(* Logix 5000 project; controller reports 1756-L63 rev 20.11; software revision 20.04; part 30 of 52 *)

        [2217].log_data[18].valid := 1, [2217].log_data[19].valid := 1, [2217].time.Year := 2023, [2217].time.Month := 1, [2217].time.Day := 17, [2217].time.Hour := 9, [2217].time.Minute := 9, [2217].time.Second := 59, [2218].log_data[0].min := 1.0, [2218].log_data[0].max := 1.0, [2218].log_data[0].total := 300.0, [2218].log_data[0].time := 300.0, [2218].log_data[0].minminute := 10, [2218].log_data[0].maxminute := 10, [2218].log_data[0].valid := 1, [2218].log_data[1].valid := 1, [2218].log_data[2].valid := 1, [2218].log_data[3].valid := 1, [2218].log_data[4].valid := 1, [2218].log_data[5].valid := 1, [2218].log_data[6].valid := 1, [2218].log_data[7].valid := 1, [2218].log_data[8].valid := 1, [2218].log_data[9].valid := 1, [2218].log_data[10].valid := 1, [2218].log_data[11].valid := 1, [2218].log_data[12].valid := 1, [2218].log_data[13].valid := 1, [2218].log_data[14].valid := 1, [2218].log_data[15].valid := 1, [2218].log_data[16].valid := 1, [2218].log_data[17].valid := 1, [2218].log_data[18].valid := 1, [2218].log_data[19].valid := 1, [2218].time.Year := 2023, [2218].time.Month := 1, [2218].time.Day := 17, [2218].time.Hour := 9, [2218].time.Minute := 14, [2218].time.Second := 59, [2219].log_data[0].min := 1.0, [2219].log_data[0].max := 1.0, [2219].log_data[0].total := 300.0, [2219].log_data[0].time := 300.0, [2219].log_data[0].minminute := 15, [2219].log_data[0].maxminute := 15, [2219].log_data[0].valid := 1, [2219].log_data[1].valid := 1, [2219].log_data[2].valid := 1, [2219].log_data[3].valid := 1, [2219].log_data[4].valid := 1, [2219].log_data[5].valid := 1, [2219].log_data[6].valid := 1, [2219].log_data[7].valid := 1, [2219].log_data[8].valid := 1, [2219].log_data[9].valid := 1, [2219].log_data[10].valid := 1, [2219].log_data[11].valid := 1, [2219].log_data[12].valid := 1, [2219].log_data[13].valid := 1,
        [2219].log_data[14].valid := 1, [2219].log_data[15].valid := 1, [2219].log_data[16].valid := 1, [2219].log_data[17].valid := 1, [2219].log_data[18].valid := 1, [2219].log_data[19].valid := 1, [2219].time.Year := 2023, [2219].time.Month := 1, [2219].time.Day := 17, [2219].time.Hour := 9, [2219].time.Minute := 19, [2219].time.Second := 59, [2220].log_data[0].min := 1.0, [2220].log_data[0].max := 1.0, [2220].log_data[0].total := 300.0, [2220].log_data[0].time := 300.0, [2220].log_data[0].minminute := 20, [2220].log_data[0].maxminute := 20, [2220].log_data[0].valid := 1, [2220].log_data[1].valid := 1, [2220].log_data[2].valid := 1, [2220].log_data[3].valid := 1, [2220].log_data[4].valid := 1, [2220].log_data[5].valid := 1, [2220].log_data[6].valid := 1, [2220].log_data[7].valid := 1, [2220].log_data[8].valid := 1, [2220].log_data[9].valid := 1, [2220].log_data[10].valid := 1, [2220].log_data[11].valid := 1, [2220].log_data[12].valid := 1, [2220].log_data[13].valid := 1, [2220].log_data[14].valid := 1, [2220].log_data[15].valid := 1, [2220].log_data[16].valid := 1, [2220].log_data[17].valid := 1, [2220].log_data[18].valid := 1, [2220].log_data[19].valid := 1, [2220].time.Year := 2023, [2220].time.Month := 1, [2220].time.Day := 17, [2220].time.Hour := 9, [2220].time.Minute := 24, [2220].time.Second := 59, [2221].log_data[0].min := 1.0, [2221].log_data[0].max := 1.0, [2221].log_data[0].total := 300.0, [2221].log_data[0].time := 300.0, [2221].log_data[0].minminute := 25, [2221].log_data[0].maxminute := 25, [2221].log_data[0].valid := 1, [2221].log_data[1].valid := 1, [2221].log_data[2].valid := 1, [2221].log_data[3].valid := 1, [2221].log_data[4].valid := 1, [2221].log_data[5].valid := 1, [2221].log_data[6].valid := 1, [2221].log_data[7].valid := 1, [2221].log_data[8].valid := 1, [2221].log_data[9].valid := 1,
        [2221].log_data[10].valid := 1, [2221].log_data[11].valid := 1, [2221].log_data[12].valid := 1, [2221].log_data[13].valid := 1, [2221].log_data[14].valid := 1, [2221].log_data[15].valid := 1, [2221].log_data[16].valid := 1, [2221].log_data[17].valid := 1, [2221].log_data[18].valid := 1, [2221].log_data[19].valid := 1, [2221].time.Year := 2023, [2221].time.Month := 1, [2221].time.Day := 17, [2221].time.Hour := 9, [2221].time.Minute := 29, [2221].time.Second := 59, [2222].log_data[0].min := 1.0, [2222].log_data[0].max := 1.0, [2222].log_data[0].total := 300.0, [2222].log_data[0].time := 300.0, [2222].log_data[0].minminute := 30, [2222].log_data[0].maxminute := 30, [2222].log_data[0].valid := 1, [2222].log_data[1].valid := 1, [2222].log_data[2].valid := 1, [2222].log_data[3].valid := 1, [2222].log_data[4].valid := 1, [2222].log_data[5].valid := 1, [2222].log_data[6].valid := 1, [2222].log_data[7].valid := 1, [2222].log_data[8].valid := 1, [2222].log_data[9].valid := 1, [2222].log_data[10].valid := 1, [2222].log_data[11].valid := 1, [2222].log_data[12].valid := 1, [2222].log_data[13].valid := 1, [2222].log_data[14].valid := 1, [2222].log_data[15].valid := 1, [2222].log_data[16].valid := 1, [2222].log_data[17].valid := 1, [2222].log_data[18].valid := 1, [2222].log_data[19].valid := 1, [2222].time.Year := 2023, [2222].time.Month := 1, [2222].time.Day := 17, [2222].time.Hour := 9, [2222].time.Minute := 34, [2222].time.Second := 59, [2223].log_data[0].min := 1.0, [2223].log_data[0].max := 1.0, [2223].log_data[0].total := 300.0, [2223].log_data[0].time := 300.0, [2223].log_data[0].minminute := 35, [2223].log_data[0].maxminute := 35, [2223].log_data[0].valid := 1, [2223].log_data[1].valid := 1, [2223].log_data[2].valid := 1, [2223].log_data[3].valid := 1, [2223].log_data[4].valid := 1, [2223].log_data[5].valid := 1,
        [2223].log_data[6].valid := 1, [2223].log_data[7].valid := 1, [2223].log_data[8].valid := 1, [2223].log_data[9].valid := 1, [2223].log_data[10].valid := 1, [2223].log_data[11].valid := 1, [2223].log_data[12].valid := 1, [2223].log_data[13].valid := 1, [2223].log_data[14].valid := 1, [2223].log_data[15].valid := 1, [2223].log_data[16].valid := 1, [2223].log_data[17].valid := 1, [2223].log_data[18].valid := 1, [2223].log_data[19].valid := 1, [2223].time.Year := 2023, [2223].time.Month := 1, [2223].time.Day := 17, [2223].time.Hour := 9, [2223].time.Minute := 39, [2223].time.Second := 59, [2224].log_data[0].min := 1.0, [2224].log_data[0].max := 1.0, [2224].log_data[0].total := 300.0, [2224].log_data[0].time := 300.0, [2224].log_data[0].minminute := 40, [2224].log_data[0].maxminute := 40, [2224].log_data[0].valid := 1, [2224].log_data[1].valid := 1, [2224].log_data[2].valid := 1, [2224].log_data[3].valid := 1, [2224].log_data[4].valid := 1, [2224].log_data[5].valid := 1, [2224].log_data[6].valid := 1, [2224].log_data[7].valid := 1, [2224].log_data[8].valid := 1, [2224].log_data[9].valid := 1, [2224].log_data[10].valid := 1, [2224].log_data[11].valid := 1, [2224].log_data[12].valid := 1, [2224].log_data[13].valid := 1, [2224].log_data[14].valid := 1, [2224].log_data[15].valid := 1, [2224].log_data[16].valid := 1, [2224].log_data[17].valid := 1, [2224].log_data[18].valid := 1, [2224].log_data[19].valid := 1, [2224].time.Year := 2023, [2224].time.Month := 1, [2224].time.Day := 17, [2224].time.Hour := 9, [2224].time.Minute := 44, [2224].time.Second := 59, [2225].log_data[0].min := 1.0, [2225].log_data[0].max := 1.0, [2225].log_data[0].total := 300.0, [2225].log_data[0].time := 300.0, [2225].log_data[0].minminute := 45, [2225].log_data[0].maxminute := 45, [2225].log_data[0].valid := 1, [2225].log_data[1].valid := 1,
        [2225].log_data[2].valid := 1, [2225].log_data[3].valid := 1, [2225].log_data[4].valid := 1, [2225].log_data[5].valid := 1, [2225].log_data[6].valid := 1, [2225].log_data[7].valid := 1, [2225].log_data[8].valid := 1, [2225].log_data[9].valid := 1, [2225].log_data[10].valid := 1, [2225].log_data[11].valid := 1, [2225].log_data[12].valid := 1, [2225].log_data[13].valid := 1, [2225].log_data[14].valid := 1, [2225].log_data[15].valid := 1, [2225].log_data[16].valid := 1, [2225].log_data[17].valid := 1, [2225].log_data[18].valid := 1, [2225].log_data[19].valid := 1, [2225].time.Year := 2023, [2225].time.Month := 1, [2225].time.Day := 17, [2225].time.Hour := 9, [2225].time.Minute := 49, [2225].time.Second := 59, [2226].log_data[0].min := 1.0, [2226].log_data[0].max := 1.0, [2226].log_data[0].total := 300.0, [2226].log_data[0].time := 300.0, [2226].log_data[0].minminute := 50, [2226].log_data[0].maxminute := 50, [2226].log_data[0].valid := 1, [2226].log_data[1].valid := 1, [2226].log_data[2].valid := 1, [2226].log_data[3].valid := 1, [2226].log_data[4].valid := 1, [2226].log_data[5].valid := 1, [2226].log_data[6].valid := 1, [2226].log_data[7].valid := 1, [2226].log_data[8].valid := 1, [2226].log_data[9].valid := 1, [2226].log_data[10].valid := 1, [2226].log_data[11].valid := 1, [2226].log_data[12].valid := 1, [2226].log_data[13].valid := 1, [2226].log_data[14].valid := 1, [2226].log_data[15].valid := 1, [2226].log_data[16].valid := 1, [2226].log_data[17].valid := 1, [2226].log_data[18].valid := 1, [2226].log_data[19].valid := 1, [2226].time.Year := 2023, [2226].time.Month := 1, [2226].time.Day := 17, [2226].time.Hour := 9, [2226].time.Minute := 54, [2226].time.Second := 59, [2227].log_data[0].min := 1.0, [2227].log_data[0].max := 1.0, [2227].log_data[0].total := 300.0, [2227].log_data[0].time := 300.0,
        [2227].log_data[0].minminute := 55, [2227].log_data[0].maxminute := 55, [2227].log_data[0].valid := 1, [2227].log_data[1].valid := 1, [2227].log_data[2].valid := 1, [2227].log_data[3].valid := 1, [2227].log_data[4].valid := 1, [2227].log_data[5].valid := 1, [2227].log_data[6].valid := 1, [2227].log_data[7].valid := 1, [2227].log_data[8].valid := 1, [2227].log_data[9].valid := 1, [2227].log_data[10].valid := 1, [2227].log_data[11].valid := 1, [2227].log_data[12].valid := 1, [2227].log_data[13].valid := 1, [2227].log_data[14].valid := 1, [2227].log_data[15].valid := 1, [2227].log_data[16].valid := 1, [2227].log_data[17].valid := 1, [2227].log_data[18].valid := 1, [2227].log_data[19].valid := 1, [2227].time.Year := 2023, [2227].time.Month := 1, [2227].time.Day := 17, [2227].time.Hour := 9, [2227].time.Minute := 59, [2227].time.Second := 59, [2228].log_data[0].min := 1.0, [2228].log_data[0].max := 1.0, [2228].log_data[0].total := 300.0, [2228].log_data[0].time := 300.0, [2228].log_data[0].valid := 1, [2228].log_data[1].valid := 1, [2228].log_data[2].valid := 1, [2228].log_data[3].valid := 1, [2228].log_data[4].valid := 1, [2228].log_data[5].valid := 1, [2228].log_data[6].valid := 1, [2228].log_data[7].valid := 1, [2228].log_data[8].valid := 1, [2228].log_data[9].valid := 1, [2228].log_data[10].valid := 1, [2228].log_data[11].valid := 1, [2228].log_data[12].valid := 1, [2228].log_data[13].valid := 1, [2228].log_data[14].valid := 1, [2228].log_data[15].valid := 1, [2228].log_data[16].valid := 1, [2228].log_data[17].valid := 1, [2228].log_data[18].valid := 1, [2228].log_data[19].valid := 1, [2228].time.Year := 2023, [2228].time.Month := 1, [2228].time.Day := 17, [2228].time.Hour := 10, [2228].time.Minute := 4, [2228].time.Second := 59, [2229].log_data[0].min := 1.0, [2229].log_data[0].max := 1.0,
        [2229].log_data[0].total := 300.0, [2229].log_data[0].time := 300.0, [2229].log_data[0].minminute := 5, [2229].log_data[0].maxminute := 5, [2229].log_data[0].valid := 1, [2229].log_data[1].valid := 1, [2229].log_data[2].valid := 1, [2229].log_data[3].valid := 1, [2229].log_data[4].valid := 1, [2229].log_data[5].valid := 1, [2229].log_data[6].valid := 1, [2229].log_data[7].valid := 1, [2229].log_data[8].valid := 1, [2229].log_data[9].valid := 1, [2229].log_data[10].valid := 1, [2229].log_data[11].valid := 1, [2229].log_data[12].valid := 1, [2229].log_data[13].valid := 1, [2229].log_data[14].valid := 1, [2229].log_data[15].valid := 1, [2229].log_data[16].valid := 1, [2229].log_data[17].valid := 1, [2229].log_data[18].valid := 1, [2229].log_data[19].valid := 1, [2229].time.Year := 2023, [2229].time.Month := 1, [2229].time.Day := 17, [2229].time.Hour := 10, [2229].time.Minute := 9, [2229].time.Second := 59, [2230].log_data[0].min := 1.0, [2230].log_data[0].max := 1.0, [2230].log_data[0].total := 300.0, [2230].log_data[0].time := 300.0, [2230].log_data[0].minminute := 10, [2230].log_data[0].maxminute := 10, [2230].log_data[0].valid := 1, [2230].log_data[1].valid := 1, [2230].log_data[2].valid := 1, [2230].log_data[3].valid := 1, [2230].log_data[4].valid := 1, [2230].log_data[5].valid := 1, [2230].log_data[6].valid := 1, [2230].log_data[7].valid := 1, [2230].log_data[8].valid := 1, [2230].log_data[9].valid := 1, [2230].log_data[10].valid := 1, [2230].log_data[11].valid := 1, [2230].log_data[12].valid := 1, [2230].log_data[13].valid := 1, [2230].log_data[14].valid := 1, [2230].log_data[15].valid := 1, [2230].log_data[16].valid := 1, [2230].log_data[17].valid := 1, [2230].log_data[18].valid := 1, [2230].log_data[19].valid := 1, [2230].time.Year := 2023, [2230].time.Month := 1, [2230].time.Day := 17, [2230].time.Hour := 10,
        [2230].time.Minute := 14, [2230].time.Second := 59, [2231].log_data[0].min := 1.0, [2231].log_data[0].max := 1.0, [2231].log_data[0].total := 300.0, [2231].log_data[0].time := 300.0, [2231].log_data[0].minminute := 15, [2231].log_data[0].maxminute := 15, [2231].log_data[0].valid := 1, [2231].log_data[1].valid := 1, [2231].log_data[2].valid := 1, [2231].log_data[3].valid := 1, [2231].log_data[4].valid := 1, [2231].log_data[5].valid := 1, [2231].log_data[6].valid := 1, [2231].log_data[7].valid := 1, [2231].log_data[8].valid := 1, [2231].log_data[9].valid := 1, [2231].log_data[10].valid := 1, [2231].log_data[11].valid := 1, [2231].log_data[12].valid := 1, [2231].log_data[13].valid := 1, [2231].log_data[14].valid := 1, [2231].log_data[15].valid := 1, [2231].log_data[16].valid := 1, [2231].log_data[17].valid := 1, [2231].log_data[18].valid := 1, [2231].log_data[19].valid := 1, [2231].time.Year := 2023, [2231].time.Month := 1, [2231].time.Day := 17, [2231].time.Hour := 10, [2231].time.Minute := 19, [2231].time.Second := 59, [2232].log_data[0].min := 1.0, [2232].log_data[0].max := 1.0, [2232].log_data[0].total := 300.0, [2232].log_data[0].time := 300.0, [2232].log_data[0].minminute := 20, [2232].log_data[0].maxminute := 20, [2232].log_data[0].valid := 1, [2232].log_data[1].valid := 1, [2232].log_data[2].valid := 1, [2232].log_data[3].valid := 1, [2232].log_data[4].valid := 1, [2232].log_data[5].valid := 1, [2232].log_data[6].valid := 1, [2232].log_data[7].valid := 1, [2232].log_data[8].valid := 1, [2232].log_data[9].valid := 1, [2232].log_data[10].valid := 1, [2232].log_data[11].valid := 1, [2232].log_data[12].valid := 1, [2232].log_data[13].valid := 1, [2232].log_data[14].valid := 1, [2232].log_data[15].valid := 1, [2232].log_data[16].valid := 1, [2232].log_data[17].valid := 1, [2232].log_data[18].valid := 1, [2232].log_data[19].valid := 1,
        [2232].time.Year := 2023, [2232].time.Month := 1, [2232].time.Day := 17, [2232].time.Hour := 10, [2232].time.Minute := 24, [2232].time.Second := 59, [2233].log_data[0].min := 1.0, [2233].log_data[0].max := 1.0, [2233].log_data[0].total := 300.0, [2233].log_data[0].time := 300.0, [2233].log_data[0].minminute := 25, [2233].log_data[0].maxminute := 25, [2233].log_data[0].valid := 1, [2233].log_data[1].valid := 1, [2233].log_data[2].valid := 1, [2233].log_data[3].valid := 1, [2233].log_data[4].valid := 1, [2233].log_data[5].valid := 1, [2233].log_data[6].valid := 1, [2233].log_data[7].valid := 1, [2233].log_data[8].valid := 1, [2233].log_data[9].valid := 1, [2233].log_data[10].valid := 1, [2233].log_data[11].valid := 1, [2233].log_data[12].valid := 1, [2233].log_data[13].valid := 1, [2233].log_data[14].valid := 1, [2233].log_data[15].valid := 1, [2233].log_data[16].valid := 1, [2233].log_data[17].valid := 1, [2233].log_data[18].valid := 1, [2233].log_data[19].valid := 1, [2233].time.Year := 2023, [2233].time.Month := 1, [2233].time.Day := 17, [2233].time.Hour := 10, [2233].time.Minute := 29, [2233].time.Second := 59, [2234].log_data[0].min := 1.0, [2234].log_data[0].max := 1.0, [2234].log_data[0].total := 300.0, [2234].log_data[0].time := 300.0, [2234].log_data[0].minminute := 30, [2234].log_data[0].maxminute := 30, [2234].log_data[0].valid := 1, [2234].log_data[1].valid := 1, [2234].log_data[2].valid := 1, [2234].log_data[3].valid := 1, [2234].log_data[4].valid := 1, [2234].log_data[5].valid := 1, [2234].log_data[6].valid := 1, [2234].log_data[7].valid := 1, [2234].log_data[8].valid := 1, [2234].log_data[9].valid := 1, [2234].log_data[10].valid := 1, [2234].log_data[11].valid := 1, [2234].log_data[12].valid := 1, [2234].log_data[13].valid := 1, [2234].log_data[14].valid := 1, [2234].log_data[15].valid := 1,
        [2234].log_data[16].valid := 1, [2234].log_data[17].valid := 1, [2234].log_data[18].valid := 1, [2234].log_data[19].valid := 1, [2234].time.Year := 2023, [2234].time.Month := 1, [2234].time.Day := 17, [2234].time.Hour := 10, [2234].time.Minute := 34, [2234].time.Second := 59, [2235].log_data[0].min := 1.0, [2235].log_data[0].max := 1.0, [2235].log_data[0].total := 300.0, [2235].log_data[0].time := 300.0, [2235].log_data[0].minminute := 35, [2235].log_data[0].maxminute := 35, [2235].log_data[0].valid := 1, [2235].log_data[1].valid := 1, [2235].log_data[2].valid := 1, [2235].log_data[3].valid := 1, [2235].log_data[4].valid := 1, [2235].log_data[5].valid := 1, [2235].log_data[6].valid := 1, [2235].log_data[7].valid := 1, [2235].log_data[8].valid := 1, [2235].log_data[9].valid := 1, [2235].log_data[10].valid := 1, [2235].log_data[11].valid := 1, [2235].log_data[12].valid := 1, [2235].log_data[13].valid := 1, [2235].log_data[14].valid := 1, [2235].log_data[15].valid := 1, [2235].log_data[16].valid := 1, [2235].log_data[17].valid := 1, [2235].log_data[18].valid := 1, [2235].log_data[19].valid := 1, [2235].time.Year := 2023, [2235].time.Month := 1, [2235].time.Day := 17, [2235].time.Hour := 10, [2235].time.Minute := 39, [2235].time.Second := 59, [2236].log_data[0].min := 1.0, [2236].log_data[0].max := 1.0, [2236].log_data[0].total := 300.0, [2236].log_data[0].time := 300.0, [2236].log_data[0].minminute := 40, [2236].log_data[0].maxminute := 40, [2236].log_data[0].valid := 1, [2236].log_data[1].valid := 1, [2236].log_data[2].valid := 1, [2236].log_data[3].valid := 1, [2236].log_data[4].valid := 1, [2236].log_data[5].valid := 1, [2236].log_data[6].valid := 1, [2236].log_data[7].valid := 1, [2236].log_data[8].valid := 1, [2236].log_data[9].valid := 1, [2236].log_data[10].valid := 1, [2236].log_data[11].valid := 1,
        [2236].log_data[12].valid := 1, [2236].log_data[13].valid := 1, [2236].log_data[14].valid := 1, [2236].log_data[15].valid := 1, [2236].log_data[16].valid := 1, [2236].log_data[17].valid := 1, [2236].log_data[18].valid := 1, [2236].log_data[19].valid := 1, [2236].time.Year := 2023, [2236].time.Month := 1, [2236].time.Day := 17, [2236].time.Hour := 10, [2236].time.Minute := 44, [2236].time.Second := 59, [2237].log_data[0].min := 1.0, [2237].log_data[0].max := 1.0, [2237].log_data[0].total := 300.0, [2237].log_data[0].time := 300.0, [2237].log_data[0].minminute := 45, [2237].log_data[0].maxminute := 45, [2237].log_data[0].valid := 1, [2237].log_data[1].valid := 1, [2237].log_data[2].valid := 1, [2237].log_data[3].valid := 1, [2237].log_data[4].valid := 1, [2237].log_data[5].valid := 1, [2237].log_data[6].valid := 1, [2237].log_data[7].valid := 1, [2237].log_data[8].valid := 1, [2237].log_data[9].valid := 1, [2237].log_data[10].valid := 1, [2237].log_data[11].valid := 1, [2237].log_data[12].valid := 1, [2237].log_data[13].valid := 1, [2237].log_data[14].valid := 1, [2237].log_data[15].valid := 1, [2237].log_data[16].valid := 1, [2237].log_data[17].valid := 1, [2237].log_data[18].valid := 1, [2237].log_data[19].valid := 1, [2237].time.Year := 2023, [2237].time.Month := 1, [2237].time.Day := 17, [2237].time.Hour := 10, [2237].time.Minute := 49, [2237].time.Second := 59, [2238].log_data[0].min := 1.0, [2238].log_data[0].max := 1.0, [2238].log_data[0].total := 300.0, [2238].log_data[0].time := 300.0, [2238].log_data[0].minminute := 50, [2238].log_data[0].maxminute := 50, [2238].log_data[0].valid := 1, [2238].log_data[1].valid := 1, [2238].log_data[2].valid := 1, [2238].log_data[3].valid := 1, [2238].log_data[4].valid := 1, [2238].log_data[5].valid := 1, [2238].log_data[6].valid := 1, [2238].log_data[7].valid := 1,
        [2238].log_data[8].valid := 1, [2238].log_data[9].valid := 1, [2238].log_data[10].valid := 1, [2238].log_data[11].valid := 1, [2238].log_data[12].valid := 1, [2238].log_data[13].valid := 1, [2238].log_data[14].valid := 1, [2238].log_data[15].valid := 1, [2238].log_data[16].valid := 1, [2238].log_data[17].valid := 1, [2238].log_data[18].valid := 1, [2238].log_data[19].valid := 1, [2238].time.Year := 2023, [2238].time.Month := 1, [2238].time.Day := 17, [2238].time.Hour := 10, [2238].time.Minute := 54, [2238].time.Second := 59, [2239].log_data[0].min := 1.0, [2239].log_data[0].max := 1.0, [2239].log_data[0].total := 300.0, [2239].log_data[0].time := 300.0, [2239].log_data[0].minminute := 55, [2239].log_data[0].maxminute := 55, [2239].log_data[0].valid := 1, [2239].log_data[1].valid := 1, [2239].log_data[2].valid := 1, [2239].log_data[3].valid := 1, [2239].log_data[4].valid := 1, [2239].log_data[5].valid := 1, [2239].log_data[6].valid := 1, [2239].log_data[7].valid := 1, [2239].log_data[8].valid := 1, [2239].log_data[9].valid := 1, [2239].log_data[10].valid := 1, [2239].log_data[11].valid := 1, [2239].log_data[12].valid := 1, [2239].log_data[13].valid := 1, [2239].log_data[14].valid := 1, [2239].log_data[15].valid := 1, [2239].log_data[16].valid := 1, [2239].log_data[17].valid := 1, [2239].log_data[18].valid := 1, [2239].log_data[19].valid := 1, [2239].time.Year := 2023, [2239].time.Month := 1, [2239].time.Day := 17, [2239].time.Hour := 10, [2239].time.Minute := 59, [2239].time.Second := 59, [2240].log_data[0].min := 1.0, [2240].log_data[0].max := 1.0, [2240].log_data[0].total := 300.0, [2240].log_data[0].time := 300.0, [2240].log_data[0].valid := 1, [2240].log_data[1].valid := 1, [2240].log_data[2].valid := 1, [2240].log_data[3].valid := 1, [2240].log_data[4].valid := 1, [2240].log_data[5].valid := 1,
        [2240].log_data[6].valid := 1, [2240].log_data[7].valid := 1, [2240].log_data[8].valid := 1, [2240].log_data[9].valid := 1, [2240].log_data[10].valid := 1, [2240].log_data[11].valid := 1, [2240].log_data[12].valid := 1, [2240].log_data[13].valid := 1, [2240].log_data[14].valid := 1, [2240].log_data[15].valid := 1, [2240].log_data[16].valid := 1, [2240].log_data[17].valid := 1, [2240].log_data[18].valid := 1, [2240].log_data[19].valid := 1, [2240].time.Year := 2023, [2240].time.Month := 1, [2240].time.Day := 17, [2240].time.Hour := 11, [2240].time.Minute := 4, [2240].time.Second := 59, [2241].log_data[0].min := 1.0, [2241].log_data[0].max := 1.0, [2241].log_data[0].total := 300.0, [2241].log_data[0].time := 300.0, [2241].log_data[0].minminute := 5, [2241].log_data[0].maxminute := 5, [2241].log_data[0].valid := 1, [2241].log_data[1].valid := 1, [2241].log_data[2].valid := 1, [2241].log_data[3].valid := 1, [2241].log_data[4].valid := 1, [2241].log_data[5].valid := 1, [2241].log_data[6].valid := 1, [2241].log_data[7].valid := 1, [2241].log_data[8].valid := 1, [2241].log_data[9].valid := 1, [2241].log_data[10].valid := 1, [2241].log_data[11].valid := 1, [2241].log_data[12].valid := 1, [2241].log_data[13].valid := 1, [2241].log_data[14].valid := 1, [2241].log_data[15].valid := 1, [2241].log_data[16].valid := 1, [2241].log_data[17].valid := 1, [2241].log_data[18].valid := 1, [2241].log_data[19].valid := 1, [2241].time.Year := 2023, [2241].time.Month := 1, [2241].time.Day := 17, [2241].time.Hour := 11, [2241].time.Minute := 9, [2241].time.Second := 59, [2242].log_data[0].min := 1.0, [2242].log_data[0].max := 1.0, [2242].log_data[0].total := 300.0, [2242].log_data[0].time := 300.0, [2242].log_data[0].minminute := 10, [2242].log_data[0].maxminute := 10, [2242].log_data[0].valid := 1, [2242].log_data[1].valid := 1,
        [2242].log_data[2].valid := 1, [2242].log_data[3].valid := 1, [2242].log_data[4].valid := 1, [2242].log_data[5].valid := 1, [2242].log_data[6].valid := 1, [2242].log_data[7].valid := 1, [2242].log_data[8].valid := 1, [2242].log_data[9].valid := 1, [2242].log_data[10].valid := 1, [2242].log_data[11].valid := 1, [2242].log_data[12].valid := 1, [2242].log_data[13].valid := 1, [2242].log_data[14].valid := 1, [2242].log_data[15].valid := 1, [2242].log_data[16].valid := 1, [2242].log_data[17].valid := 1, [2242].log_data[18].valid := 1, [2242].log_data[19].valid := 1, [2242].time.Year := 2023, [2242].time.Month := 1, [2242].time.Day := 17, [2242].time.Hour := 11, [2242].time.Minute := 14, [2242].time.Second := 59, [2243].log_data[0].min := 1.0, [2243].log_data[0].max := 1.0, [2243].log_data[0].total := 300.0, [2243].log_data[0].time := 300.0, [2243].log_data[0].minminute := 15, [2243].log_data[0].maxminute := 15, [2243].log_data[0].valid := 1, [2243].log_data[1].valid := 1, [2243].log_data[2].valid := 1, [2243].log_data[3].valid := 1, [2243].log_data[4].valid := 1, [2243].log_data[5].valid := 1, [2243].log_data[6].valid := 1, [2243].log_data[7].valid := 1, [2243].log_data[8].valid := 1, [2243].log_data[9].valid := 1, [2243].log_data[10].valid := 1, [2243].log_data[11].valid := 1, [2243].log_data[12].valid := 1, [2243].log_data[13].valid := 1, [2243].log_data[14].valid := 1, [2243].log_data[15].valid := 1, [2243].log_data[16].valid := 1, [2243].log_data[17].valid := 1, [2243].log_data[18].valid := 1, [2243].log_data[19].valid := 1, [2243].time.Year := 2023, [2243].time.Month := 1, [2243].time.Day := 17, [2243].time.Hour := 11, [2243].time.Minute := 19, [2243].time.Second := 59, [2244].log_data[0].min := 1.0, [2244].log_data[0].max := 1.0, [2244].log_data[0].total := 300.0, [2244].log_data[0].time := 300.0,
        [2244].log_data[0].minminute := 20, [2244].log_data[0].maxminute := 20, [2244].log_data[0].valid := 1, [2244].log_data[1].valid := 1, [2244].log_data[2].valid := 1, [2244].log_data[3].valid := 1, [2244].log_data[4].valid := 1, [2244].log_data[5].valid := 1, [2244].log_data[6].valid := 1, [2244].log_data[7].valid := 1, [2244].log_data[8].valid := 1, [2244].log_data[9].valid := 1, [2244].log_data[10].valid := 1, [2244].log_data[11].valid := 1, [2244].log_data[12].valid := 1, [2244].log_data[13].valid := 1, [2244].log_data[14].valid := 1, [2244].log_data[15].valid := 1, [2244].log_data[16].valid := 1, [2244].log_data[17].valid := 1, [2244].log_data[18].valid := 1, [2244].log_data[19].valid := 1, [2244].time.Year := 2023, [2244].time.Month := 1, [2244].time.Day := 17, [2244].time.Hour := 11, [2244].time.Minute := 24, [2244].time.Second := 59, [2245].log_data[0].min := 1.0, [2245].log_data[0].max := 1.0, [2245].log_data[0].total := 300.0, [2245].log_data[0].time := 300.0, [2245].log_data[0].minminute := 25, [2245].log_data[0].maxminute := 25, [2245].log_data[0].valid := 1, [2245].log_data[1].valid := 1, [2245].log_data[2].valid := 1, [2245].log_data[3].valid := 1, [2245].log_data[4].valid := 1, [2245].log_data[5].valid := 1, [2245].log_data[6].valid := 1, [2245].log_data[7].valid := 1, [2245].log_data[8].valid := 1, [2245].log_data[9].valid := 1, [2245].log_data[10].valid := 1, [2245].log_data[11].valid := 1, [2245].log_data[12].valid := 1, [2245].log_data[13].valid := 1, [2245].log_data[14].valid := 1, [2245].log_data[15].valid := 1, [2245].log_data[16].valid := 1, [2245].log_data[17].valid := 1, [2245].log_data[18].valid := 1, [2245].log_data[19].valid := 1, [2245].time.Year := 2023, [2245].time.Month := 1, [2245].time.Day := 17, [2245].time.Hour := 11, [2245].time.Minute := 29, [2245].time.Second := 59,
        [2246].log_data[0].min := 1.0, [2246].log_data[0].max := 1.0, [2246].log_data[0].total := 300.0, [2246].log_data[0].time := 300.0, [2246].log_data[0].minminute := 30, [2246].log_data[0].maxminute := 30, [2246].log_data[0].valid := 1, [2246].log_data[1].valid := 1, [2246].log_data[2].valid := 1, [2246].log_data[3].valid := 1, [2246].log_data[4].valid := 1, [2246].log_data[5].valid := 1, [2246].log_data[6].valid := 1, [2246].log_data[7].valid := 1, [2246].log_data[8].valid := 1, [2246].log_data[9].valid := 1, [2246].log_data[10].valid := 1, [2246].log_data[11].valid := 1, [2246].log_data[12].valid := 1, [2246].log_data[13].valid := 1, [2246].log_data[14].valid := 1, [2246].log_data[15].valid := 1, [2246].log_data[16].valid := 1, [2246].log_data[17].valid := 1, [2246].log_data[18].valid := 1, [2246].log_data[19].valid := 1, [2246].time.Year := 2023, [2246].time.Month := 1, [2246].time.Day := 17, [2246].time.Hour := 11, [2246].time.Minute := 34, [2246].time.Second := 59, [2247].log_data[0].min := 1.0, [2247].log_data[0].max := 1.0, [2247].log_data[0].total := 300.0, [2247].log_data[0].time := 300.0, [2247].log_data[0].minminute := 35, [2247].log_data[0].maxminute := 35, [2247].log_data[0].valid := 1, [2247].log_data[1].valid := 1, [2247].log_data[2].valid := 1, [2247].log_data[3].valid := 1, [2247].log_data[4].valid := 1, [2247].log_data[5].valid := 1, [2247].log_data[6].valid := 1, [2247].log_data[7].valid := 1, [2247].log_data[8].valid := 1, [2247].log_data[9].valid := 1, [2247].log_data[10].valid := 1, [2247].log_data[11].valid := 1, [2247].log_data[12].valid := 1, [2247].log_data[13].valid := 1, [2247].log_data[14].valid := 1, [2247].log_data[15].valid := 1, [2247].log_data[16].valid := 1, [2247].log_data[17].valid := 1, [2247].log_data[18].valid := 1, [2247].log_data[19].valid := 1, [2247].time.Year := 2023, [2247].time.Month := 1,
        [2247].time.Day := 17, [2247].time.Hour := 11, [2247].time.Minute := 39, [2247].time.Second := 59, [2248].log_data[0].min := 1.0, [2248].log_data[0].max := 1.0, [2248].log_data[0].total := 300.0, [2248].log_data[0].time := 300.0, [2248].log_data[0].minminute := 40, [2248].log_data[0].maxminute := 40, [2248].log_data[0].valid := 1, [2248].log_data[1].valid := 1, [2248].log_data[2].valid := 1, [2248].log_data[3].valid := 1, [2248].log_data[4].valid := 1, [2248].log_data[5].valid := 1, [2248].log_data[6].valid := 1, [2248].log_data[7].valid := 1, [2248].log_data[8].valid := 1, [2248].log_data[9].valid := 1, [2248].log_data[10].valid := 1, [2248].log_data[11].valid := 1, [2248].log_data[12].valid := 1, [2248].log_data[13].valid := 1, [2248].log_data[14].valid := 1, [2248].log_data[15].valid := 1, [2248].log_data[16].valid := 1, [2248].log_data[17].valid := 1, [2248].log_data[18].valid := 1, [2248].log_data[19].valid := 1, [2248].time.Year := 2023, [2248].time.Month := 1, [2248].time.Day := 17, [2248].time.Hour := 11, [2248].time.Minute := 44, [2248].time.Second := 59, [2249].log_data[0].min := 1.0, [2249].log_data[0].max := 1.0, [2249].log_data[0].total := 300.0, [2249].log_data[0].time := 300.0, [2249].log_data[0].minminute := 45, [2249].log_data[0].maxminute := 45, [2249].log_data[0].valid := 1, [2249].log_data[1].valid := 1, [2249].log_data[2].valid := 1, [2249].log_data[3].valid := 1, [2249].log_data[4].valid := 1, [2249].log_data[5].valid := 1, [2249].log_data[6].valid := 1, [2249].log_data[7].valid := 1, [2249].log_data[8].valid := 1, [2249].log_data[9].valid := 1, [2249].log_data[10].valid := 1, [2249].log_data[11].valid := 1, [2249].log_data[12].valid := 1, [2249].log_data[13].valid := 1, [2249].log_data[14].valid := 1, [2249].log_data[15].valid := 1, [2249].log_data[16].valid := 1, [2249].log_data[17].valid := 1,
        [2249].log_data[18].valid := 1, [2249].log_data[19].valid := 1, [2249].time.Year := 2023, [2249].time.Month := 1, [2249].time.Day := 17, [2249].time.Hour := 11, [2249].time.Minute := 49, [2249].time.Second := 59, [2250].log_data[0].min := 1.0, [2250].log_data[0].max := 1.0, [2250].log_data[0].total := 300.0, [2250].log_data[0].time := 300.0, [2250].log_data[0].minminute := 50, [2250].log_data[0].maxminute := 50, [2250].log_data[0].valid := 1, [2250].log_data[1].valid := 1, [2250].log_data[2].valid := 1, [2250].log_data[3].valid := 1, [2250].log_data[4].valid := 1, [2250].log_data[5].valid := 1, [2250].log_data[6].valid := 1, [2250].log_data[7].valid := 1, [2250].log_data[8].valid := 1, [2250].log_data[9].valid := 1, [2250].log_data[10].valid := 1, [2250].log_data[11].valid := 1, [2250].log_data[12].valid := 1, [2250].log_data[13].valid := 1, [2250].log_data[14].valid := 1, [2250].log_data[15].valid := 1, [2250].log_data[16].valid := 1, [2250].log_data[17].valid := 1, [2250].log_data[18].valid := 1, [2250].log_data[19].valid := 1, [2250].time.Year := 2023, [2250].time.Month := 1, [2250].time.Day := 17, [2250].time.Hour := 11, [2250].time.Minute := 54, [2250].time.Second := 59, [2251].log_data[0].min := 1.0, [2251].log_data[0].max := 1.0, [2251].log_data[0].total := 300.0, [2251].log_data[0].time := 300.0, [2251].log_data[0].minminute := 55, [2251].log_data[0].maxminute := 55, [2251].log_data[0].valid := 1, [2251].log_data[1].valid := 1, [2251].log_data[2].valid := 1, [2251].log_data[3].valid := 1, [2251].log_data[4].valid := 1, [2251].log_data[5].valid := 1, [2251].log_data[6].valid := 1, [2251].log_data[7].valid := 1, [2251].log_data[8].valid := 1, [2251].log_data[9].valid := 1, [2251].log_data[10].valid := 1, [2251].log_data[11].valid := 1, [2251].log_data[12].valid := 1, [2251].log_data[13].valid := 1,
        [2251].log_data[14].valid := 1, [2251].log_data[15].valid := 1, [2251].log_data[16].valid := 1, [2251].log_data[17].valid := 1, [2251].log_data[18].valid := 1, [2251].log_data[19].valid := 1, [2251].time.Year := 2023, [2251].time.Month := 1, [2251].time.Day := 17, [2251].time.Hour := 11, [2251].time.Minute := 59, [2251].time.Second := 59, [2252].log_data[0].min := 1.0, [2252].log_data[0].max := 1.0, [2252].log_data[0].total := 300.0, [2252].log_data[0].time := 300.0, [2252].log_data[0].valid := 1, [2252].log_data[1].valid := 1, [2252].log_data[2].valid := 1, [2252].log_data[3].valid := 1, [2252].log_data[4].valid := 1, [2252].log_data[5].valid := 1, [2252].log_data[6].valid := 1, [2252].log_data[7].valid := 1, [2252].log_data[8].valid := 1, [2252].log_data[9].valid := 1, [2252].log_data[10].valid := 1, [2252].log_data[11].valid := 1, [2252].log_data[12].valid := 1, [2252].log_data[13].valid := 1, [2252].log_data[14].valid := 1, [2252].log_data[15].valid := 1, [2252].log_data[16].valid := 1, [2252].log_data[17].valid := 1, [2252].log_data[18].valid := 1, [2252].log_data[19].valid := 1, [2252].time.Year := 2023, [2252].time.Month := 1, [2252].time.Day := 17, [2252].time.Hour := 12, [2252].time.Minute := 4, [2252].time.Second := 59, [2253].log_data[0].min := 1.0, [2253].log_data[0].max := 1.0, [2253].log_data[0].total := 300.0, [2253].log_data[0].time := 300.0, [2253].log_data[0].minminute := 5, [2253].log_data[0].maxminute := 5, [2253].log_data[0].valid := 1, [2253].log_data[1].valid := 1, [2253].log_data[2].valid := 1, [2253].log_data[3].valid := 1, [2253].log_data[4].valid := 1, [2253].log_data[5].valid := 1, [2253].log_data[6].valid := 1, [2253].log_data[7].valid := 1, [2253].log_data[8].valid := 1, [2253].log_data[9].valid := 1, [2253].log_data[10].valid := 1, [2253].log_data[11].valid := 1,
        [2253].log_data[12].valid := 1, [2253].log_data[13].valid := 1, [2253].log_data[14].valid := 1, [2253].log_data[15].valid := 1, [2253].log_data[16].valid := 1, [2253].log_data[17].valid := 1, [2253].log_data[18].valid := 1, [2253].log_data[19].valid := 1, [2253].time.Year := 2023, [2253].time.Month := 1, [2253].time.Day := 17, [2253].time.Hour := 12, [2253].time.Minute := 9, [2253].time.Second := 59, [2254].log_data[0].min := 1.0, [2254].log_data[0].max := 1.0, [2254].log_data[0].total := 300.0, [2254].log_data[0].time := 300.0, [2254].log_data[0].minminute := 10, [2254].log_data[0].maxminute := 10, [2254].log_data[0].valid := 1, [2254].log_data[1].valid := 1, [2254].log_data[2].valid := 1, [2254].log_data[3].valid := 1, [2254].log_data[4].valid := 1, [2254].log_data[5].valid := 1, [2254].log_data[6].valid := 1, [2254].log_data[7].valid := 1, [2254].log_data[8].valid := 1, [2254].log_data[9].valid := 1, [2254].log_data[10].valid := 1, [2254].log_data[11].valid := 1, [2254].log_data[12].valid := 1, [2254].log_data[13].valid := 1, [2254].log_data[14].valid := 1, [2254].log_data[15].valid := 1, [2254].log_data[16].valid := 1, [2254].log_data[17].valid := 1, [2254].log_data[18].valid := 1, [2254].log_data[19].valid := 1, [2254].time.Year := 2023, [2254].time.Month := 1, [2254].time.Day := 17, [2254].time.Hour := 12, [2254].time.Minute := 14, [2254].time.Second := 59, [2255].log_data[0].min := 1.0, [2255].log_data[0].max := 1.0, [2255].log_data[0].total := 300.0, [2255].log_data[0].time := 300.0, [2255].log_data[0].minminute := 15, [2255].log_data[0].maxminute := 15, [2255].log_data[0].valid := 1, [2255].log_data[1].valid := 1, [2255].log_data[2].valid := 1, [2255].log_data[3].valid := 1, [2255].log_data[4].valid := 1, [2255].log_data[5].valid := 1, [2255].log_data[6].valid := 1, [2255].log_data[7].valid := 1,
        [2255].log_data[8].valid := 1, [2255].log_data[9].valid := 1, [2255].log_data[10].valid := 1, [2255].log_data[11].valid := 1, [2255].log_data[12].valid := 1, [2255].log_data[13].valid := 1, [2255].log_data[14].valid := 1, [2255].log_data[15].valid := 1, [2255].log_data[16].valid := 1, [2255].log_data[17].valid := 1, [2255].log_data[18].valid := 1, [2255].log_data[19].valid := 1, [2255].time.Year := 2023, [2255].time.Month := 1, [2255].time.Day := 17, [2255].time.Hour := 12, [2255].time.Minute := 19, [2255].time.Second := 59, [2256].log_data[0].min := 1.0, [2256].log_data[0].max := 1.0, [2256].log_data[0].total := 300.0, [2256].log_data[0].time := 300.0, [2256].log_data[0].minminute := 20, [2256].log_data[0].maxminute := 20, [2256].log_data[0].valid := 1, [2256].log_data[1].valid := 1, [2256].log_data[2].valid := 1, [2256].log_data[3].valid := 1, [2256].log_data[4].valid := 1, [2256].log_data[5].valid := 1, [2256].log_data[6].valid := 1, [2256].log_data[7].valid := 1, [2256].log_data[8].valid := 1, [2256].log_data[9].valid := 1, [2256].log_data[10].valid := 1, [2256].log_data[11].valid := 1, [2256].log_data[12].valid := 1, [2256].log_data[13].valid := 1, [2256].log_data[14].valid := 1, [2256].log_data[15].valid := 1, [2256].log_data[16].valid := 1, [2256].log_data[17].valid := 1, [2256].log_data[18].valid := 1, [2256].log_data[19].valid := 1, [2256].time.Year := 2023, [2256].time.Month := 1, [2256].time.Day := 17, [2256].time.Hour := 12, [2256].time.Minute := 24, [2256].time.Second := 59, [2257].log_data[0].min := 1.0, [2257].log_data[0].max := 1.0, [2257].log_data[0].total := 300.0, [2257].log_data[0].time := 300.0, [2257].log_data[0].minminute := 25, [2257].log_data[0].maxminute := 25, [2257].log_data[0].valid := 1, [2257].log_data[1].valid := 1, [2257].log_data[2].valid := 1, [2257].log_data[3].valid := 1,
        [2257].log_data[4].valid := 1, [2257].log_data[5].valid := 1, [2257].log_data[6].valid := 1, [2257].log_data[7].valid := 1, [2257].log_data[8].valid := 1, [2257].log_data[9].valid := 1, [2257].log_data[10].valid := 1, [2257].log_data[11].valid := 1, [2257].log_data[12].valid := 1, [2257].log_data[13].valid := 1, [2257].log_data[14].valid := 1, [2257].log_data[15].valid := 1, [2257].log_data[16].valid := 1, [2257].log_data[17].valid := 1, [2257].log_data[18].valid := 1, [2257].log_data[19].valid := 1, [2257].time.Year := 2023, [2257].time.Month := 1, [2257].time.Day := 17, [2257].time.Hour := 12, [2257].time.Minute := 29, [2257].time.Second := 59, [2258].log_data[0].min := 1.0, [2258].log_data[0].max := 1.0, [2258].log_data[0].total := 300.0, [2258].log_data[0].time := 300.0, [2258].log_data[0].minminute := 30, [2258].log_data[0].maxminute := 30, [2258].log_data[0].valid := 1, [2258].log_data[1].valid := 1, [2258].log_data[2].valid := 1, [2258].log_data[3].valid := 1, [2258].log_data[4].valid := 1, [2258].log_data[5].valid := 1, [2258].log_data[6].valid := 1, [2258].log_data[7].valid := 1, [2258].log_data[8].valid := 1, [2258].log_data[9].valid := 1, [2258].log_data[10].valid := 1, [2258].log_data[11].valid := 1, [2258].log_data[12].valid := 1, [2258].log_data[13].valid := 1, [2258].log_data[14].valid := 1, [2258].log_data[15].valid := 1, [2258].log_data[16].valid := 1, [2258].log_data[17].valid := 1, [2258].log_data[18].valid := 1, [2258].log_data[19].valid := 1, [2258].time.Year := 2023, [2258].time.Month := 1, [2258].time.Day := 17, [2258].time.Hour := 12, [2258].time.Minute := 34, [2258].time.Second := 59, [2259].log_data[0].min := 1.0, [2259].log_data[0].max := 1.0, [2259].log_data[0].total := 300.0, [2259].log_data[0].time := 300.0, [2259].log_data[0].minminute := 35, [2259].log_data[0].maxminute := 35,
        [2259].log_data[0].valid := 1, [2259].log_data[1].valid := 1, [2259].log_data[2].valid := 1, [2259].log_data[3].valid := 1, [2259].log_data[4].valid := 1, [2259].log_data[5].valid := 1, [2259].log_data[6].valid := 1, [2259].log_data[7].valid := 1, [2259].log_data[8].valid := 1, [2259].log_data[9].valid := 1, [2259].log_data[10].valid := 1, [2259].log_data[11].valid := 1, [2259].log_data[12].valid := 1, [2259].log_data[13].valid := 1, [2259].log_data[14].valid := 1, [2259].log_data[15].valid := 1, [2259].log_data[16].valid := 1, [2259].log_data[17].valid := 1, [2259].log_data[18].valid := 1, [2259].log_data[19].valid := 1, [2259].time.Year := 2023, [2259].time.Month := 1, [2259].time.Day := 17, [2259].time.Hour := 12, [2259].time.Minute := 39, [2259].time.Second := 59, [2260].log_data[0].min := 1.0, [2260].log_data[0].max := 1.0, [2260].log_data[0].total := 300.0, [2260].log_data[0].time := 300.0, [2260].log_data[0].minminute := 40, [2260].log_data[0].maxminute := 40, [2260].log_data[0].valid := 1, [2260].log_data[1].valid := 1, [2260].log_data[2].valid := 1, [2260].log_data[3].valid := 1, [2260].log_data[4].valid := 1, [2260].log_data[5].valid := 1, [2260].log_data[6].valid := 1, [2260].log_data[7].valid := 1, [2260].log_data[8].valid := 1, [2260].log_data[9].valid := 1, [2260].log_data[10].valid := 1, [2260].log_data[11].valid := 1, [2260].log_data[12].valid := 1, [2260].log_data[13].valid := 1, [2260].log_data[14].valid := 1, [2260].log_data[15].valid := 1, [2260].log_data[16].valid := 1, [2260].log_data[17].valid := 1, [2260].log_data[18].valid := 1, [2260].log_data[19].valid := 1, [2260].time.Year := 2023, [2260].time.Month := 1, [2260].time.Day := 17, [2260].time.Hour := 12, [2260].time.Minute := 44, [2260].time.Second := 59, [2261].log_data[0].min := 1.0, [2261].log_data[0].max := 1.0,
        [2261].log_data[0].total := 300.0, [2261].log_data[0].time := 300.0, [2261].log_data[0].minminute := 45, [2261].log_data[0].maxminute := 45, [2261].log_data[0].valid := 1, [2261].log_data[1].valid := 1, [2261].log_data[2].valid := 1, [2261].log_data[3].valid := 1, [2261].log_data[4].valid := 1, [2261].log_data[5].valid := 1, [2261].log_data[6].valid := 1, [2261].log_data[7].valid := 1, [2261].log_data[8].valid := 1, [2261].log_data[9].valid := 1, [2261].log_data[10].valid := 1, [2261].log_data[11].valid := 1, [2261].log_data[12].valid := 1, [2261].log_data[13].valid := 1, [2261].log_data[14].valid := 1, [2261].log_data[15].valid := 1, [2261].log_data[16].valid := 1, [2261].log_data[17].valid := 1, [2261].log_data[18].valid := 1, [2261].log_data[19].valid := 1, [2261].time.Year := 2023, [2261].time.Month := 1, [2261].time.Day := 17, [2261].time.Hour := 12, [2261].time.Minute := 49, [2261].time.Second := 59, [2262].log_data[0].min := 1.0, [2262].log_data[0].max := 1.0, [2262].log_data[0].total := 300.0, [2262].log_data[0].time := 300.0, [2262].log_data[0].minminute := 50, [2262].log_data[0].maxminute := 50, [2262].log_data[0].valid := 1, [2262].log_data[1].valid := 1, [2262].log_data[2].valid := 1, [2262].log_data[3].valid := 1, [2262].log_data[4].valid := 1, [2262].log_data[5].valid := 1, [2262].log_data[6].valid := 1, [2262].log_data[7].valid := 1, [2262].log_data[8].valid := 1, [2262].log_data[9].valid := 1, [2262].log_data[10].valid := 1, [2262].log_data[11].valid := 1, [2262].log_data[12].valid := 1, [2262].log_data[13].valid := 1, [2262].log_data[14].valid := 1, [2262].log_data[15].valid := 1, [2262].log_data[16].valid := 1, [2262].log_data[17].valid := 1, [2262].log_data[18].valid := 1, [2262].log_data[19].valid := 1, [2262].time.Year := 2023, [2262].time.Month := 1, [2262].time.Day := 17, [2262].time.Hour := 12,
        [2262].time.Minute := 54, [2262].time.Second := 59, [2263].log_data[0].min := 1.0, [2263].log_data[0].max := 1.0, [2263].log_data[0].total := 300.0, [2263].log_data[0].time := 300.0, [2263].log_data[0].minminute := 55, [2263].log_data[0].maxminute := 55, [2263].log_data[0].valid := 1, [2263].log_data[1].valid := 1, [2263].log_data[2].valid := 1, [2263].log_data[3].valid := 1, [2263].log_data[4].valid := 1, [2263].log_data[5].valid := 1, [2263].log_data[6].valid := 1, [2263].log_data[7].valid := 1, [2263].log_data[8].valid := 1, [2263].log_data[9].valid := 1, [2263].log_data[10].valid := 1, [2263].log_data[11].valid := 1, [2263].log_data[12].valid := 1, [2263].log_data[13].valid := 1, [2263].log_data[14].valid := 1, [2263].log_data[15].valid := 1, [2263].log_data[16].valid := 1, [2263].log_data[17].valid := 1, [2263].log_data[18].valid := 1, [2263].log_data[19].valid := 1, [2263].time.Year := 2023, [2263].time.Month := 1, [2263].time.Day := 17, [2263].time.Hour := 12, [2263].time.Minute := 59, [2263].time.Second := 59, [2264].log_data[0].min := 1.0, [2264].log_data[0].max := 1.0, [2264].log_data[0].total := 300.0, [2264].log_data[0].time := 300.0, [2264].log_data[0].valid := 1, [2264].log_data[1].valid := 1, [2264].log_data[2].valid := 1, [2264].log_data[3].valid := 1, [2264].log_data[4].valid := 1, [2264].log_data[5].valid := 1, [2264].log_data[6].valid := 1, [2264].log_data[7].valid := 1, [2264].log_data[8].valid := 1, [2264].log_data[9].valid := 1, [2264].log_data[10].valid := 1, [2264].log_data[11].valid := 1, [2264].log_data[12].valid := 1, [2264].log_data[13].valid := 1, [2264].log_data[14].valid := 1, [2264].log_data[15].valid := 1, [2264].log_data[16].valid := 1, [2264].log_data[17].valid := 1, [2264].log_data[18].valid := 1, [2264].log_data[19].valid := 1, [2264].time.Year := 2023, [2264].time.Month := 1,
        [2264].time.Day := 17, [2264].time.Hour := 13, [2264].time.Minute := 4, [2264].time.Second := 59, [2265].log_data[0].min := 1.0, [2265].log_data[0].max := 1.0, [2265].log_data[0].total := 300.0, [2265].log_data[0].time := 300.0, [2265].log_data[0].minminute := 5, [2265].log_data[0].maxminute := 5, [2265].log_data[0].valid := 1, [2265].log_data[1].valid := 1, [2265].log_data[2].valid := 1, [2265].log_data[3].valid := 1, [2265].log_data[4].valid := 1, [2265].log_data[5].valid := 1, [2265].log_data[6].valid := 1, [2265].log_data[7].valid := 1, [2265].log_data[8].valid := 1, [2265].log_data[9].valid := 1, [2265].log_data[10].valid := 1, [2265].log_data[11].valid := 1, [2265].log_data[12].valid := 1, [2265].log_data[13].valid := 1, [2265].log_data[14].valid := 1, [2265].log_data[15].valid := 1, [2265].log_data[16].valid := 1, [2265].log_data[17].valid := 1, [2265].log_data[18].valid := 1, [2265].log_data[19].valid := 1, [2265].time.Year := 2023, [2265].time.Month := 1, [2265].time.Day := 17, [2265].time.Hour := 13, [2265].time.Minute := 9, [2265].time.Second := 59, [2266].log_data[0].min := 1.0, [2266].log_data[0].max := 1.0, [2266].log_data[0].total := 300.0, [2266].log_data[0].time := 300.0, [2266].log_data[0].minminute := 10, [2266].log_data[0].maxminute := 10, [2266].log_data[0].valid := 1, [2266].log_data[1].valid := 1, [2266].log_data[2].valid := 1, [2266].log_data[3].valid := 1, [2266].log_data[4].valid := 1, [2266].log_data[5].valid := 1, [2266].log_data[6].valid := 1, [2266].log_data[7].valid := 1, [2266].log_data[8].valid := 1, [2266].log_data[9].valid := 1, [2266].log_data[10].valid := 1, [2266].log_data[11].valid := 1, [2266].log_data[12].valid := 1, [2266].log_data[13].valid := 1, [2266].log_data[14].valid := 1, [2266].log_data[15].valid := 1, [2266].log_data[16].valid := 1, [2266].log_data[17].valid := 1,
        [2266].log_data[18].valid := 1, [2266].log_data[19].valid := 1, [2266].time.Year := 2023, [2266].time.Month := 1, [2266].time.Day := 17, [2266].time.Hour := 13, [2266].time.Minute := 14, [2266].time.Second := 59, [2267].log_data[0].min := 1.0, [2267].log_data[0].max := 1.0, [2267].log_data[0].total := 300.0, [2267].log_data[0].time := 300.0, [2267].log_data[0].minminute := 15, [2267].log_data[0].maxminute := 15, [2267].log_data[0].valid := 1, [2267].log_data[1].valid := 1, [2267].log_data[2].valid := 1, [2267].log_data[3].valid := 1, [2267].log_data[4].valid := 1, [2267].log_data[5].valid := 1, [2267].log_data[6].valid := 1, [2267].log_data[7].valid := 1, [2267].log_data[8].valid := 1, [2267].log_data[9].valid := 1, [2267].log_data[10].valid := 1, [2267].log_data[11].valid := 1, [2267].log_data[12].valid := 1, [2267].log_data[13].valid := 1, [2267].log_data[14].valid := 1, [2267].log_data[15].valid := 1, [2267].log_data[16].valid := 1, [2267].log_data[17].valid := 1, [2267].log_data[18].valid := 1, [2267].log_data[19].valid := 1, [2267].time.Year := 2023, [2267].time.Month := 1, [2267].time.Day := 17, [2267].time.Hour := 13, [2267].time.Minute := 19, [2267].time.Second := 59, [2268].log_data[0].min := 1.0, [2268].log_data[0].max := 1.0, [2268].log_data[0].total := 300.0, [2268].log_data[0].time := 300.0, [2268].log_data[0].minminute := 20, [2268].log_data[0].maxminute := 20, [2268].log_data[0].valid := 1, [2268].log_data[1].valid := 1, [2268].log_data[2].valid := 1, [2268].log_data[3].valid := 1, [2268].log_data[4].valid := 1, [2268].log_data[5].valid := 1, [2268].log_data[6].valid := 1, [2268].log_data[7].valid := 1, [2268].log_data[8].valid := 1, [2268].log_data[9].valid := 1, [2268].log_data[10].valid := 1, [2268].log_data[11].valid := 1, [2268].log_data[12].valid := 1, [2268].log_data[13].valid := 1,
        [2268].log_data[14].valid := 1, [2268].log_data[15].valid := 1, [2268].log_data[16].valid := 1, [2268].log_data[17].valid := 1, [2268].log_data[18].valid := 1, [2268].log_data[19].valid := 1, [2268].time.Year := 2023, [2268].time.Month := 1, [2268].time.Day := 17, [2268].time.Hour := 13, [2268].time.Minute := 24, [2268].time.Second := 59, [2269].log_data[0].min := 1.0, [2269].log_data[0].max := 1.0, [2269].log_data[0].total := 300.0, [2269].log_data[0].time := 300.0, [2269].log_data[0].minminute := 25, [2269].log_data[0].maxminute := 25, [2269].log_data[0].valid := 1, [2269].log_data[1].valid := 1, [2269].log_data[2].valid := 1, [2269].log_data[3].valid := 1, [2269].log_data[4].valid := 1, [2269].log_data[5].valid := 1, [2269].log_data[6].valid := 1, [2269].log_data[7].valid := 1, [2269].log_data[8].valid := 1, [2269].log_data[9].valid := 1, [2269].log_data[10].valid := 1, [2269].log_data[11].valid := 1, [2269].log_data[12].valid := 1, [2269].log_data[13].valid := 1, [2269].log_data[14].valid := 1, [2269].log_data[15].valid := 1, [2269].log_data[16].valid := 1, [2269].log_data[17].valid := 1, [2269].log_data[18].valid := 1, [2269].log_data[19].valid := 1, [2269].time.Year := 2023, [2269].time.Month := 1, [2269].time.Day := 17, [2269].time.Hour := 13, [2269].time.Minute := 29, [2269].time.Second := 59, [2270].log_data[0].min := 1.0, [2270].log_data[0].max := 1.0, [2270].log_data[0].total := 300.0, [2270].log_data[0].time := 300.0, [2270].log_data[0].minminute := 30, [2270].log_data[0].maxminute := 30, [2270].log_data[0].valid := 1, [2270].log_data[1].valid := 1, [2270].log_data[2].valid := 1, [2270].log_data[3].valid := 1, [2270].log_data[4].valid := 1, [2270].log_data[5].valid := 1, [2270].log_data[6].valid := 1, [2270].log_data[7].valid := 1, [2270].log_data[8].valid := 1, [2270].log_data[9].valid := 1,
        [2270].log_data[10].valid := 1, [2270].log_data[11].valid := 1, [2270].log_data[12].valid := 1, [2270].log_data[13].valid := 1, [2270].log_data[14].valid := 1, [2270].log_data[15].valid := 1, [2270].log_data[16].valid := 1, [2270].log_data[17].valid := 1, [2270].log_data[18].valid := 1, [2270].log_data[19].valid := 1, [2270].time.Year := 2023, [2270].time.Month := 1, [2270].time.Day := 17, [2270].time.Hour := 13, [2270].time.Minute := 34, [2270].time.Second := 59, [2271].log_data[0].min := 1.0, [2271].log_data[0].max := 1.0, [2271].log_data[0].total := 300.0, [2271].log_data[0].time := 300.0, [2271].log_data[0].minminute := 35, [2271].log_data[0].maxminute := 35, [2271].log_data[0].valid := 1, [2271].log_data[1].valid := 1, [2271].log_data[2].valid := 1, [2271].log_data[3].valid := 1, [2271].log_data[4].valid := 1, [2271].log_data[5].valid := 1, [2271].log_data[6].valid := 1, [2271].log_data[7].valid := 1, [2271].log_data[8].valid := 1, [2271].log_data[9].valid := 1, [2271].log_data[10].valid := 1, [2271].log_data[11].valid := 1, [2271].log_data[12].valid := 1, [2271].log_data[13].valid := 1, [2271].log_data[14].valid := 1, [2271].log_data[15].valid := 1, [2271].log_data[16].valid := 1, [2271].log_data[17].valid := 1, [2271].log_data[18].valid := 1, [2271].log_data[19].valid := 1, [2271].time.Year := 2023, [2271].time.Month := 1, [2271].time.Day := 17, [2271].time.Hour := 13, [2271].time.Minute := 39, [2271].time.Second := 59, [2272].log_data[0].min := 1.0, [2272].log_data[0].max := 1.0, [2272].log_data[0].total := 300.0, [2272].log_data[0].time := 300.0, [2272].log_data[0].minminute := 40, [2272].log_data[0].maxminute := 40, [2272].log_data[0].valid := 1, [2272].log_data[1].valid := 1, [2272].log_data[2].valid := 1, [2272].log_data[3].valid := 1, [2272].log_data[4].valid := 1, [2272].log_data[5].valid := 1,
        [2272].log_data[6].valid := 1, [2272].log_data[7].valid := 1, [2272].log_data[8].valid := 1, [2272].log_data[9].valid := 1, [2272].log_data[10].valid := 1, [2272].log_data[11].valid := 1, [2272].log_data[12].valid := 1, [2272].log_data[13].valid := 1, [2272].log_data[14].valid := 1, [2272].log_data[15].valid := 1, [2272].log_data[16].valid := 1, [2272].log_data[17].valid := 1, [2272].log_data[18].valid := 1, [2272].log_data[19].valid := 1, [2272].time.Year := 2023, [2272].time.Month := 1, [2272].time.Day := 17, [2272].time.Hour := 13, [2272].time.Minute := 44, [2272].time.Second := 59, [2273].log_data[0].min := 1.0, [2273].log_data[0].max := 1.0, [2273].log_data[0].total := 300.0, [2273].log_data[0].time := 300.0, [2273].log_data[0].minminute := 45, [2273].log_data[0].maxminute := 45, [2273].log_data[0].valid := 1, [2273].log_data[1].valid := 1, [2273].log_data[2].valid := 1, [2273].log_data[3].valid := 1, [2273].log_data[4].valid := 1, [2273].log_data[5].valid := 1, [2273].log_data[6].valid := 1, [2273].log_data[7].valid := 1, [2273].log_data[8].valid := 1, [2273].log_data[9].valid := 1, [2273].log_data[10].valid := 1, [2273].log_data[11].valid := 1, [2273].log_data[12].valid := 1, [2273].log_data[13].valid := 1, [2273].log_data[14].valid := 1, [2273].log_data[15].valid := 1, [2273].log_data[16].valid := 1, [2273].log_data[17].valid := 1, [2273].log_data[18].valid := 1, [2273].log_data[19].valid := 1, [2273].time.Year := 2023, [2273].time.Month := 1, [2273].time.Day := 17, [2273].time.Hour := 13, [2273].time.Minute := 49, [2273].time.Second := 59, [2274].log_data[0].min := 1.0, [2274].log_data[0].max := 1.0, [2274].log_data[0].total := 300.0, [2274].log_data[0].time := 300.0, [2274].log_data[0].minminute := 50, [2274].log_data[0].maxminute := 50, [2274].log_data[0].valid := 1, [2274].log_data[1].valid := 1,
        [2274].log_data[2].valid := 1, [2274].log_data[3].valid := 1, [2274].log_data[4].valid := 1, [2274].log_data[5].valid := 1, [2274].log_data[6].valid := 1, [2274].log_data[7].valid := 1, [2274].log_data[8].valid := 1, [2274].log_data[9].valid := 1, [2274].log_data[10].valid := 1, [2274].log_data[11].valid := 1, [2274].log_data[12].valid := 1, [2274].log_data[13].valid := 1, [2274].log_data[14].valid := 1, [2274].log_data[15].valid := 1, [2274].log_data[16].valid := 1, [2274].log_data[17].valid := 1, [2274].log_data[18].valid := 1, [2274].log_data[19].valid := 1, [2274].time.Year := 2023, [2274].time.Month := 1, [2274].time.Day := 17, [2274].time.Hour := 13, [2274].time.Minute := 54, [2274].time.Second := 59, [2275].log_data[0].min := 1.0, [2275].log_data[0].max := 1.0, [2275].log_data[0].total := 300.0, [2275].log_data[0].time := 300.0, [2275].log_data[0].minminute := 55, [2275].log_data[0].maxminute := 55, [2275].log_data[0].valid := 1, [2275].log_data[1].valid := 1, [2275].log_data[2].valid := 1, [2275].log_data[3].valid := 1, [2275].log_data[4].valid := 1, [2275].log_data[5].valid := 1, [2275].log_data[6].valid := 1, [2275].log_data[7].valid := 1, [2275].log_data[8].valid := 1, [2275].log_data[9].valid := 1, [2275].log_data[10].valid := 1, [2275].log_data[11].valid := 1, [2275].log_data[12].valid := 1, [2275].log_data[13].valid := 1, [2275].log_data[14].valid := 1, [2275].log_data[15].valid := 1, [2275].log_data[16].valid := 1, [2275].log_data[17].valid := 1, [2275].log_data[18].valid := 1, [2275].log_data[19].valid := 1, [2275].time.Year := 2023, [2275].time.Month := 1, [2275].time.Day := 17, [2275].time.Hour := 13, [2275].time.Minute := 59, [2275].time.Second := 59, [2276].log_data[0].min := 1.0, [2276].log_data[0].max := 1.0, [2276].log_data[0].total := 300.0, [2276].log_data[0].time := 300.0,
        [2276].log_data[0].valid := 1, [2276].log_data[1].valid := 1, [2276].log_data[2].valid := 1, [2276].log_data[3].valid := 1, [2276].log_data[4].valid := 1, [2276].log_data[5].valid := 1, [2276].log_data[6].valid := 1, [2276].log_data[7].valid := 1, [2276].log_data[8].valid := 1, [2276].log_data[9].valid := 1, [2276].log_data[10].valid := 1, [2276].log_data[11].valid := 1, [2276].log_data[12].valid := 1, [2276].log_data[13].valid := 1, [2276].log_data[14].valid := 1, [2276].log_data[15].valid := 1, [2276].log_data[16].valid := 1, [2276].log_data[17].valid := 1, [2276].log_data[18].valid := 1, [2276].log_data[19].valid := 1, [2276].time.Year := 2023, [2276].time.Month := 1, [2276].time.Day := 17, [2276].time.Hour := 14, [2276].time.Minute := 4, [2276].time.Second := 59, [2277].log_data[0].min := 1.0, [2277].log_data[0].max := 1.0, [2277].log_data[0].total := 300.0, [2277].log_data[0].time := 300.0, [2277].log_data[0].minminute := 5, [2277].log_data[0].maxminute := 5, [2277].log_data[0].valid := 1, [2277].log_data[1].valid := 1, [2277].log_data[2].valid := 1, [2277].log_data[3].valid := 1, [2277].log_data[4].valid := 1, [2277].log_data[5].valid := 1, [2277].log_data[6].valid := 1, [2277].log_data[7].valid := 1, [2277].log_data[8].valid := 1, [2277].log_data[9].valid := 1, [2277].log_data[10].valid := 1, [2277].log_data[11].valid := 1, [2277].log_data[12].valid := 1, [2277].log_data[13].valid := 1, [2277].log_data[14].valid := 1, [2277].log_data[15].valid := 1, [2277].log_data[16].valid := 1, [2277].log_data[17].valid := 1, [2277].log_data[18].valid := 1, [2277].log_data[19].valid := 1, [2277].time.Year := 2023, [2277].time.Month := 1, [2277].time.Day := 17, [2277].time.Hour := 14, [2277].time.Minute := 9, [2277].time.Second := 59, [2278].log_data[0].min := 1.0, [2278].log_data[0].max := 1.0,
        [2278].log_data[0].total := 300.0, [2278].log_data[0].time := 300.0, [2278].log_data[0].minminute := 10, [2278].log_data[0].maxminute := 10, [2278].log_data[0].valid := 1, [2278].log_data[1].valid := 1, [2278].log_data[2].valid := 1, [2278].log_data[3].valid := 1, [2278].log_data[4].valid := 1, [2278].log_data[5].valid := 1, [2278].log_data[6].valid := 1, [2278].log_data[7].valid := 1, [2278].log_data[8].valid := 1, [2278].log_data[9].valid := 1, [2278].log_data[10].valid := 1, [2278].log_data[11].valid := 1, [2278].log_data[12].valid := 1, [2278].log_data[13].valid := 1, [2278].log_data[14].valid := 1, [2278].log_data[15].valid := 1, [2278].log_data[16].valid := 1, [2278].log_data[17].valid := 1, [2278].log_data[18].valid := 1, [2278].log_data[19].valid := 1, [2278].time.Year := 2023, [2278].time.Month := 1, [2278].time.Day := 17, [2278].time.Hour := 14, [2278].time.Minute := 14, [2278].time.Second := 59, [2279].log_data[0].min := 1.0, [2279].log_data[0].max := 1.0, [2279].log_data[0].total := 300.0, [2279].log_data[0].time := 300.0, [2279].log_data[0].minminute := 15, [2279].log_data[0].maxminute := 15, [2279].log_data[0].valid := 1, [2279].log_data[1].valid := 1, [2279].log_data[2].valid := 1, [2279].log_data[3].valid := 1, [2279].log_data[4].valid := 1, [2279].log_data[5].valid := 1, [2279].log_data[6].valid := 1, [2279].log_data[7].valid := 1, [2279].log_data[8].valid := 1, [2279].log_data[9].valid := 1, [2279].log_data[10].valid := 1, [2279].log_data[11].valid := 1, [2279].log_data[12].valid := 1, [2279].log_data[13].valid := 1, [2279].log_data[14].valid := 1, [2279].log_data[15].valid := 1, [2279].log_data[16].valid := 1, [2279].log_data[17].valid := 1, [2279].log_data[18].valid := 1, [2279].log_data[19].valid := 1, [2279].time.Year := 2023, [2279].time.Month := 1, [2279].time.Day := 17, [2279].time.Hour := 14,
        [2279].time.Minute := 19, [2279].time.Second := 59, [2280].log_data[0].min := 1.0, [2280].log_data[0].max := 1.0, [2280].log_data[0].total := 300.0, [2280].log_data[0].time := 300.0, [2280].log_data[0].minminute := 20, [2280].log_data[0].maxminute := 20, [2280].log_data[0].valid := 1, [2280].log_data[1].valid := 1, [2280].log_data[2].valid := 1, [2280].log_data[3].valid := 1, [2280].log_data[4].valid := 1, [2280].log_data[5].valid := 1, [2280].log_data[6].valid := 1, [2280].log_data[7].valid := 1, [2280].log_data[8].valid := 1, [2280].log_data[9].valid := 1, [2280].log_data[10].valid := 1, [2280].log_data[11].valid := 1, [2280].log_data[12].valid := 1, [2280].log_data[13].valid := 1, [2280].log_data[14].valid := 1, [2280].log_data[15].valid := 1, [2280].log_data[16].valid := 1, [2280].log_data[17].valid := 1, [2280].log_data[18].valid := 1, [2280].log_data[19].valid := 1, [2280].time.Year := 2023, [2280].time.Month := 1, [2280].time.Day := 17, [2280].time.Hour := 14, [2280].time.Minute := 24, [2280].time.Second := 59, [2281].log_data[0].min := 1.0, [2281].log_data[0].max := 1.0, [2281].log_data[0].total := 300.0, [2281].log_data[0].time := 300.0, [2281].log_data[0].minminute := 25, [2281].log_data[0].maxminute := 25, [2281].log_data[0].valid := 1, [2281].log_data[1].valid := 1, [2281].log_data[2].valid := 1, [2281].log_data[3].valid := 1, [2281].log_data[4].valid := 1, [2281].log_data[5].valid := 1, [2281].log_data[6].valid := 1, [2281].log_data[7].valid := 1, [2281].log_data[8].valid := 1, [2281].log_data[9].valid := 1, [2281].log_data[10].valid := 1, [2281].log_data[11].valid := 1, [2281].log_data[12].valid := 1, [2281].log_data[13].valid := 1, [2281].log_data[14].valid := 1, [2281].log_data[15].valid := 1, [2281].log_data[16].valid := 1, [2281].log_data[17].valid := 1, [2281].log_data[18].valid := 1, [2281].log_data[19].valid := 1,
        [2281].time.Year := 2023, [2281].time.Month := 1, [2281].time.Day := 17, [2281].time.Hour := 14, [2281].time.Minute := 29, [2281].time.Second := 59, [2282].log_data[0].min := 1.0, [2282].log_data[0].max := 1.0, [2282].log_data[0].total := 300.0, [2282].log_data[0].time := 300.0, [2282].log_data[0].minminute := 30, [2282].log_data[0].maxminute := 30, [2282].log_data[0].valid := 1, [2282].log_data[1].valid := 1, [2282].log_data[2].valid := 1, [2282].log_data[3].valid := 1, [2282].log_data[4].valid := 1, [2282].log_data[5].valid := 1, [2282].log_data[6].valid := 1, [2282].log_data[7].valid := 1, [2282].log_data[8].valid := 1, [2282].log_data[9].valid := 1, [2282].log_data[10].valid := 1, [2282].log_data[11].valid := 1, [2282].log_data[12].valid := 1, [2282].log_data[13].valid := 1, [2282].log_data[14].valid := 1, [2282].log_data[15].valid := 1, [2282].log_data[16].valid := 1, [2282].log_data[17].valid := 1, [2282].log_data[18].valid := 1, [2282].log_data[19].valid := 1, [2282].time.Year := 2023, [2282].time.Month := 1, [2282].time.Day := 17, [2282].time.Hour := 14, [2282].time.Minute := 34, [2282].time.Second := 59, [2283].log_data[0].min := 1.0, [2283].log_data[0].max := 1.0, [2283].log_data[0].total := 300.0, [2283].log_data[0].time := 300.0, [2283].log_data[0].minminute := 35, [2283].log_data[0].maxminute := 35, [2283].log_data[0].valid := 1, [2283].log_data[1].valid := 1, [2283].log_data[2].valid := 1, [2283].log_data[3].valid := 1, [2283].log_data[4].valid := 1, [2283].log_data[5].valid := 1, [2283].log_data[6].valid := 1, [2283].log_data[7].valid := 1, [2283].log_data[8].valid := 1, [2283].log_data[9].valid := 1, [2283].log_data[10].valid := 1, [2283].log_data[11].valid := 1, [2283].log_data[12].valid := 1, [2283].log_data[13].valid := 1, [2283].log_data[14].valid := 1, [2283].log_data[15].valid := 1,
        [2283].log_data[16].valid := 1, [2283].log_data[17].valid := 1, [2283].log_data[18].valid := 1, [2283].log_data[19].valid := 1, [2283].time.Year := 2023, [2283].time.Month := 1, [2283].time.Day := 17, [2283].time.Hour := 14, [2283].time.Minute := 39, [2283].time.Second := 59, [2284].log_data[0].min := 1.0, [2284].log_data[0].max := 1.0, [2284].log_data[0].total := 300.0, [2284].log_data[0].time := 300.0, [2284].log_data[0].minminute := 40, [2284].log_data[0].maxminute := 40, [2284].log_data[0].valid := 1, [2284].log_data[1].valid := 1, [2284].log_data[2].valid := 1, [2284].log_data[3].valid := 1, [2284].log_data[4].valid := 1, [2284].log_data[5].valid := 1, [2284].log_data[6].valid := 1, [2284].log_data[7].valid := 1, [2284].log_data[8].valid := 1, [2284].log_data[9].valid := 1, [2284].log_data[10].valid := 1, [2284].log_data[11].valid := 1, [2284].log_data[12].valid := 1, [2284].log_data[13].valid := 1, [2284].log_data[14].valid := 1, [2284].log_data[15].valid := 1, [2284].log_data[16].valid := 1, [2284].log_data[17].valid := 1, [2284].log_data[18].valid := 1, [2284].log_data[19].valid := 1, [2284].time.Year := 2023, [2284].time.Month := 1, [2284].time.Day := 17, [2284].time.Hour := 14, [2284].time.Minute := 44, [2284].time.Second := 59, [2285].log_data[0].min := 1.0, [2285].log_data[0].max := 1.0, [2285].log_data[0].total := 300.0, [2285].log_data[0].time := 300.0, [2285].log_data[0].minminute := 45, [2285].log_data[0].maxminute := 45, [2285].log_data[0].valid := 1, [2285].log_data[1].valid := 1, [2285].log_data[2].valid := 1, [2285].log_data[3].valid := 1, [2285].log_data[4].valid := 1, [2285].log_data[5].valid := 1, [2285].log_data[6].valid := 1, [2285].log_data[7].valid := 1, [2285].log_data[8].valid := 1, [2285].log_data[9].valid := 1, [2285].log_data[10].valid := 1, [2285].log_data[11].valid := 1,
        [2285].log_data[12].valid := 1, [2285].log_data[13].valid := 1, [2285].log_data[14].valid := 1, [2285].log_data[15].valid := 1, [2285].log_data[16].valid := 1, [2285].log_data[17].valid := 1, [2285].log_data[18].valid := 1, [2285].log_data[19].valid := 1, [2285].time.Year := 2023, [2285].time.Month := 1, [2285].time.Day := 17, [2285].time.Hour := 14, [2285].time.Minute := 49, [2285].time.Second := 59, [2286].log_data[0].min := 1.0, [2286].log_data[0].max := 1.0, [2286].log_data[0].total := 300.0, [2286].log_data[0].time := 300.0, [2286].log_data[0].minminute := 50, [2286].log_data[0].maxminute := 50, [2286].log_data[0].valid := 1, [2286].log_data[1].valid := 1, [2286].log_data[2].valid := 1, [2286].log_data[3].valid := 1, [2286].log_data[4].valid := 1, [2286].log_data[5].valid := 1, [2286].log_data[6].valid := 1, [2286].log_data[7].valid := 1, [2286].log_data[8].valid := 1, [2286].log_data[9].valid := 1, [2286].log_data[10].valid := 1, [2286].log_data[11].valid := 1, [2286].log_data[12].valid := 1, [2286].log_data[13].valid := 1, [2286].log_data[14].valid := 1, [2286].log_data[15].valid := 1, [2286].log_data[16].valid := 1, [2286].log_data[17].valid := 1, [2286].log_data[18].valid := 1, [2286].log_data[19].valid := 1, [2286].time.Year := 2023, [2286].time.Month := 1, [2286].time.Day := 17, [2286].time.Hour := 14, [2286].time.Minute := 54, [2286].time.Second := 59, [2287].log_data[0].min := 1.0, [2287].log_data[0].max := 1.0, [2287].log_data[0].total := 300.0, [2287].log_data[0].time := 300.0, [2287].log_data[0].minminute := 55, [2287].log_data[0].maxminute := 55, [2287].log_data[0].valid := 1, [2287].log_data[1].valid := 1, [2287].log_data[2].valid := 1, [2287].log_data[3].valid := 1, [2287].log_data[4].valid := 1, [2287].log_data[5].valid := 1, [2287].log_data[6].valid := 1, [2287].log_data[7].valid := 1,
        [2287].log_data[8].valid := 1, [2287].log_data[9].valid := 1, [2287].log_data[10].valid := 1, [2287].log_data[11].valid := 1, [2287].log_data[12].valid := 1, [2287].log_data[13].valid := 1, [2287].log_data[14].valid := 1, [2287].log_data[15].valid := 1, [2287].log_data[16].valid := 1, [2287].log_data[17].valid := 1, [2287].log_data[18].valid := 1, [2287].log_data[19].valid := 1, [2287].time.Year := 2023, [2287].time.Month := 1, [2287].time.Day := 17, [2287].time.Hour := 14, [2287].time.Minute := 59, [2287].time.Second := 59, [2288].log_data[0].min := 1.0, [2288].log_data[0].max := 1.0, [2288].log_data[0].total := 300.0, [2288].log_data[0].time := 300.0, [2288].log_data[0].valid := 1, [2288].log_data[1].valid := 1, [2288].log_data[2].valid := 1, [2288].log_data[3].valid := 1, [2288].log_data[4].valid := 1, [2288].log_data[5].valid := 1, [2288].log_data[6].valid := 1, [2288].log_data[7].valid := 1, [2288].log_data[8].valid := 1, [2288].log_data[9].valid := 1, [2288].log_data[10].valid := 1, [2288].log_data[11].valid := 1, [2288].log_data[12].valid := 1, [2288].log_data[13].valid := 1, [2288].log_data[14].valid := 1, [2288].log_data[15].valid := 1, [2288].log_data[16].valid := 1, [2288].log_data[17].valid := 1, [2288].log_data[18].valid := 1, [2288].log_data[19].valid := 1, [2288].time.Year := 2023, [2288].time.Month := 1, [2288].time.Day := 17, [2288].time.Hour := 15, [2288].time.Minute := 4, [2288].time.Second := 59, [2289].log_data[0].min := 1.0, [2289].log_data[0].max := 1.0, [2289].log_data[0].total := 300.0, [2289].log_data[0].time := 300.0, [2289].log_data[0].minminute := 5, [2289].log_data[0].maxminute := 5, [2289].log_data[0].valid := 1, [2289].log_data[1].valid := 1, [2289].log_data[2].valid := 1, [2289].log_data[3].valid := 1, [2289].log_data[4].valid := 1, [2289].log_data[5].valid := 1,
        [2289].log_data[6].valid := 1, [2289].log_data[7].valid := 1, [2289].log_data[8].valid := 1, [2289].log_data[9].valid := 1, [2289].log_data[10].valid := 1, [2289].log_data[11].valid := 1, [2289].log_data[12].valid := 1, [2289].log_data[13].valid := 1, [2289].log_data[14].valid := 1, [2289].log_data[15].valid := 1, [2289].log_data[16].valid := 1, [2289].log_data[17].valid := 1, [2289].log_data[18].valid := 1, [2289].log_data[19].valid := 1, [2289].time.Year := 2023, [2289].time.Month := 1, [2289].time.Day := 17, [2289].time.Hour := 15, [2289].time.Minute := 9, [2289].time.Second := 59, [2290].log_data[0].min := 1.0, [2290].log_data[0].max := 1.0, [2290].log_data[0].total := 300.0, [2290].log_data[0].time := 300.0, [2290].log_data[0].minminute := 10, [2290].log_data[0].maxminute := 10, [2290].log_data[0].valid := 1, [2290].log_data[1].valid := 1, [2290].log_data[2].valid := 1, [2290].log_data[3].valid := 1, [2290].log_data[4].valid := 1, [2290].log_data[5].valid := 1, [2290].log_data[6].valid := 1, [2290].log_data[7].valid := 1, [2290].log_data[8].valid := 1, [2290].log_data[9].valid := 1, [2290].log_data[10].valid := 1, [2290].log_data[11].valid := 1, [2290].log_data[12].valid := 1, [2290].log_data[13].valid := 1, [2290].log_data[14].valid := 1, [2290].log_data[15].valid := 1, [2290].log_data[16].valid := 1, [2290].log_data[17].valid := 1, [2290].log_data[18].valid := 1, [2290].log_data[19].valid := 1, [2290].time.Year := 2023, [2290].time.Month := 1, [2290].time.Day := 17, [2290].time.Hour := 15, [2290].time.Minute := 14, [2290].time.Second := 59, [2291].log_data[0].min := 1.0, [2291].log_data[0].max := 1.0, [2291].log_data[0].total := 300.0, [2291].log_data[0].time := 300.0, [2291].log_data[0].minminute := 15, [2291].log_data[0].maxminute := 15, [2291].log_data[0].valid := 1, [2291].log_data[1].valid := 1,
        [2291].log_data[2].valid := 1, [2291].log_data[3].valid := 1, [2291].log_data[4].valid := 1, [2291].log_data[5].valid := 1, [2291].log_data[6].valid := 1, [2291].log_data[7].valid := 1, [2291].log_data[8].valid := 1, [2291].log_data[9].valid := 1, [2291].log_data[10].valid := 1, [2291].log_data[11].valid := 1, [2291].log_data[12].valid := 1, [2291].log_data[13].valid := 1, [2291].log_data[14].valid := 1, [2291].log_data[15].valid := 1, [2291].log_data[16].valid := 1, [2291].log_data[17].valid := 1, [2291].log_data[18].valid := 1, [2291].log_data[19].valid := 1, [2291].time.Year := 2023, [2291].time.Month := 1, [2291].time.Day := 17, [2291].time.Hour := 15, [2291].time.Minute := 19, [2291].time.Second := 59, [2292].log_data[0].min := 1.0, [2292].log_data[0].max := 1.0, [2292].log_data[0].total := 300.0, [2292].log_data[0].time := 300.0, [2292].log_data[0].minminute := 20, [2292].log_data[0].maxminute := 20, [2292].log_data[0].valid := 1, [2292].log_data[1].valid := 1, [2292].log_data[2].valid := 1, [2292].log_data[3].valid := 1, [2292].log_data[4].valid := 1, [2292].log_data[5].valid := 1, [2292].log_data[6].valid := 1, [2292].log_data[7].valid := 1, [2292].log_data[8].valid := 1, [2292].log_data[9].valid := 1, [2292].log_data[10].valid := 1, [2292].log_data[11].valid := 1, [2292].log_data[12].valid := 1, [2292].log_data[13].valid := 1, [2292].log_data[14].valid := 1, [2292].log_data[15].valid := 1, [2292].log_data[16].valid := 1, [2292].log_data[17].valid := 1, [2292].log_data[18].valid := 1, [2292].log_data[19].valid := 1, [2292].time.Year := 2023, [2292].time.Month := 1, [2292].time.Day := 17, [2292].time.Hour := 15, [2292].time.Minute := 24, [2292].time.Second := 59, [2293].log_data[0].min := 1.0, [2293].log_data[0].max := 1.0, [2293].log_data[0].total := 300.0, [2293].log_data[0].time := 300.0,
        [2293].log_data[0].minminute := 25, [2293].log_data[0].maxminute := 25, [2293].log_data[0].valid := 1, [2293].log_data[1].valid := 1, [2293].log_data[2].valid := 1, [2293].log_data[3].valid := 1, [2293].log_data[4].valid := 1, [2293].log_data[5].valid := 1, [2293].log_data[6].valid := 1, [2293].log_data[7].valid := 1, [2293].log_data[8].valid := 1, [2293].log_data[9].valid := 1, [2293].log_data[10].valid := 1, [2293].log_data[11].valid := 1, [2293].log_data[12].valid := 1, [2293].log_data[13].valid := 1, [2293].log_data[14].valid := 1, [2293].log_data[15].valid := 1, [2293].log_data[16].valid := 1, [2293].log_data[17].valid := 1, [2293].log_data[18].valid := 1, [2293].log_data[19].valid := 1, [2293].time.Year := 2023, [2293].time.Month := 1, [2293].time.Day := 17, [2293].time.Hour := 15, [2293].time.Minute := 29, [2293].time.Second := 59, [2294].log_data[0].min := 1.0, [2294].log_data[0].max := 1.0, [2294].log_data[0].total := 300.0, [2294].log_data[0].time := 300.0, [2294].log_data[0].minminute := 30, [2294].log_data[0].maxminute := 30, [2294].log_data[0].valid := 1, [2294].log_data[1].valid := 1, [2294].log_data[2].valid := 1, [2294].log_data[3].valid := 1, [2294].log_data[4].valid := 1, [2294].log_data[5].valid := 1, [2294].log_data[6].valid := 1, [2294].log_data[7].valid := 1, [2294].log_data[8].valid := 1, [2294].log_data[9].valid := 1, [2294].log_data[10].valid := 1, [2294].log_data[11].valid := 1, [2294].log_data[12].valid := 1, [2294].log_data[13].valid := 1, [2294].log_data[14].valid := 1, [2294].log_data[15].valid := 1, [2294].log_data[16].valid := 1, [2294].log_data[17].valid := 1, [2294].log_data[18].valid := 1, [2294].log_data[19].valid := 1, [2294].time.Year := 2023, [2294].time.Month := 1, [2294].time.Day := 17, [2294].time.Hour := 15, [2294].time.Minute := 34, [2294].time.Second := 59,
        [2295].log_data[0].min := 1.0, [2295].log_data[0].max := 1.0, [2295].log_data[0].total := 300.0, [2295].log_data[0].time := 300.0, [2295].log_data[0].minminute := 35, [2295].log_data[0].maxminute := 35, [2295].log_data[0].valid := 1, [2295].log_data[1].valid := 1, [2295].log_data[2].valid := 1, [2295].log_data[3].valid := 1, [2295].log_data[4].valid := 1, [2295].log_data[5].valid := 1, [2295].log_data[6].valid := 1, [2295].log_data[7].valid := 1, [2295].log_data[8].valid := 1, [2295].log_data[9].valid := 1, [2295].log_data[10].valid := 1, [2295].log_data[11].valid := 1, [2295].log_data[12].valid := 1, [2295].log_data[13].valid := 1, [2295].log_data[14].valid := 1, [2295].log_data[15].valid := 1, [2295].log_data[16].valid := 1, [2295].log_data[17].valid := 1, [2295].log_data[18].valid := 1, [2295].log_data[19].valid := 1, [2295].time.Year := 2023, [2295].time.Month := 1, [2295].time.Day := 17, [2295].time.Hour := 15, [2295].time.Minute := 39, [2295].time.Second := 59, [2296].log_data[0].min := 1.0, [2296].log_data[0].max := 1.0, [2296].log_data[0].total := 300.0, [2296].log_data[0].time := 300.0, [2296].log_data[0].minminute := 40, [2296].log_data[0].maxminute := 40, [2296].log_data[0].valid := 1, [2296].log_data[1].valid := 1, [2296].log_data[2].valid := 1, [2296].log_data[3].valid := 1, [2296].log_data[4].valid := 1, [2296].log_data[5].valid := 1, [2296].log_data[6].valid := 1, [2296].log_data[7].valid := 1, [2296].log_data[8].valid := 1, [2296].log_data[9].valid := 1, [2296].log_data[10].valid := 1, [2296].log_data[11].valid := 1, [2296].log_data[12].valid := 1, [2296].log_data[13].valid := 1, [2296].log_data[14].valid := 1, [2296].log_data[15].valid := 1, [2296].log_data[16].valid := 1, [2296].log_data[17].valid := 1, [2296].log_data[18].valid := 1, [2296].log_data[19].valid := 1, [2296].time.Year := 2023, [2296].time.Month := 1,
        [2296].time.Day := 17, [2296].time.Hour := 15, [2296].time.Minute := 44, [2296].time.Second := 59, [2297].log_data[0].min := 1.0, [2297].log_data[0].max := 1.0, [2297].log_data[0].total := 300.0, [2297].log_data[0].time := 300.0, [2297].log_data[0].minminute := 45, [2297].log_data[0].maxminute := 45, [2297].log_data[0].valid := 1, [2297].log_data[1].valid := 1, [2297].log_data[2].valid := 1, [2297].log_data[3].valid := 1, [2297].log_data[4].valid := 1, [2297].log_data[5].valid := 1, [2297].log_data[6].valid := 1, [2297].log_data[7].valid := 1, [2297].log_data[8].valid := 1, [2297].log_data[9].valid := 1, [2297].log_data[10].valid := 1, [2297].log_data[11].valid := 1, [2297].log_data[12].valid := 1, [2297].log_data[13].valid := 1, [2297].log_data[14].valid := 1, [2297].log_data[15].valid := 1, [2297].log_data[16].valid := 1, [2297].log_data[17].valid := 1, [2297].log_data[18].valid := 1, [2297].log_data[19].valid := 1, [2297].time.Year := 2023, [2297].time.Month := 1, [2297].time.Day := 17, [2297].time.Hour := 15, [2297].time.Minute := 49, [2297].time.Second := 59, [2298].log_data[0].min := 1.0, [2298].log_data[0].max := 1.0, [2298].log_data[0].total := 300.0, [2298].log_data[0].time := 300.0, [2298].log_data[0].minminute := 50, [2298].log_data[0].maxminute := 50, [2298].log_data[0].valid := 1, [2298].log_data[1].valid := 1, [2298].log_data[2].valid := 1, [2298].log_data[3].valid := 1, [2298].log_data[4].valid := 1, [2298].log_data[5].valid := 1, [2298].log_data[6].valid := 1, [2298].log_data[7].valid := 1, [2298].log_data[8].valid := 1, [2298].log_data[9].valid := 1, [2298].log_data[10].valid := 1, [2298].log_data[11].valid := 1, [2298].log_data[12].valid := 1, [2298].log_data[13].valid := 1, [2298].log_data[14].valid := 1, [2298].log_data[15].valid := 1, [2298].log_data[16].valid := 1, [2298].log_data[17].valid := 1,
        [2298].log_data[18].valid := 1, [2298].log_data[19].valid := 1, [2298].time.Year := 2023, [2298].time.Month := 1, [2298].time.Day := 17, [2298].time.Hour := 15, [2298].time.Minute := 54, [2298].time.Second := 59, [2299].log_data[0].min := 1.0, [2299].log_data[0].max := 1.0, [2299].log_data[0].total := 300.0, [2299].log_data[0].time := 300.0, [2299].log_data[0].minminute := 55, [2299].log_data[0].maxminute := 55, [2299].log_data[0].valid := 1, [2299].log_data[1].valid := 1, [2299].log_data[2].valid := 1, [2299].log_data[3].valid := 1, [2299].log_data[4].valid := 1, [2299].log_data[5].valid := 1, [2299].log_data[6].valid := 1, [2299].log_data[7].valid := 1, [2299].log_data[8].valid := 1, [2299].log_data[9].valid := 1, [2299].log_data[10].valid := 1, [2299].log_data[11].valid := 1, [2299].log_data[12].valid := 1, [2299].log_data[13].valid := 1, [2299].log_data[14].valid := 1, [2299].log_data[15].valid := 1, [2299].log_data[16].valid := 1, [2299].log_data[17].valid := 1, [2299].log_data[18].valid := 1, [2299].log_data[19].valid := 1, [2299].time.Year := 2023, [2299].time.Month := 1, [2299].time.Day := 17, [2299].time.Hour := 15, [2299].time.Minute := 59, [2299].time.Second := 59, [2300].log_data[0].min := 1.0, [2300].log_data[0].max := 1.0, [2300].log_data[0].total := 300.0, [2300].log_data[0].time := 300.0, [2300].log_data[0].valid := 1, [2300].log_data[1].valid := 1, [2300].log_data[2].valid := 1, [2300].log_data[3].valid := 1, [2300].log_data[4].valid := 1, [2300].log_data[5].valid := 1, [2300].log_data[6].valid := 1, [2300].log_data[7].valid := 1, [2300].log_data[8].valid := 1, [2300].log_data[9].valid := 1, [2300].log_data[10].valid := 1, [2300].log_data[11].valid := 1, [2300].log_data[12].valid := 1, [2300].log_data[13].valid := 1, [2300].log_data[14].valid := 1, [2300].log_data[15].valid := 1,
        [2300].log_data[16].valid := 1, [2300].log_data[17].valid := 1, [2300].log_data[18].valid := 1, [2300].log_data[19].valid := 1, [2300].time.Year := 2023, [2300].time.Month := 1, [2300].time.Day := 17, [2300].time.Hour := 16, [2300].time.Minute := 4, [2300].time.Second := 59, [2301].log_data[0].min := 1.0, [2301].log_data[0].max := 1.0, [2301].log_data[0].total := 300.0, [2301].log_data[0].time := 300.0, [2301].log_data[0].minminute := 5, [2301].log_data[0].maxminute := 5, [2301].log_data[0].valid := 1, [2301].log_data[1].valid := 1, [2301].log_data[2].valid := 1, [2301].log_data[3].valid := 1, [2301].log_data[4].valid := 1, [2301].log_data[5].valid := 1, [2301].log_data[6].valid := 1, [2301].log_data[7].valid := 1, [2301].log_data[8].valid := 1, [2301].log_data[9].valid := 1, [2301].log_data[10].valid := 1, [2301].log_data[11].valid := 1, [2301].log_data[12].valid := 1, [2301].log_data[13].valid := 1, [2301].log_data[14].valid := 1, [2301].log_data[15].valid := 1, [2301].log_data[16].valid := 1, [2301].log_data[17].valid := 1, [2301].log_data[18].valid := 1, [2301].log_data[19].valid := 1, [2301].time.Year := 2023, [2301].time.Month := 1, [2301].time.Day := 17, [2301].time.Hour := 16, [2301].time.Minute := 9, [2301].time.Second := 59, [2302].log_data[0].min := 1.0, [2302].log_data[0].max := 1.0, [2302].log_data[0].total := 300.0, [2302].log_data[0].time := 300.0, [2302].log_data[0].minminute := 10, [2302].log_data[0].maxminute := 10, [2302].log_data[0].valid := 1, [2302].log_data[1].valid := 1, [2302].log_data[2].valid := 1, [2302].log_data[3].valid := 1, [2302].log_data[4].valid := 1, [2302].log_data[5].valid := 1, [2302].log_data[6].valid := 1, [2302].log_data[7].valid := 1, [2302].log_data[8].valid := 1, [2302].log_data[9].valid := 1, [2302].log_data[10].valid := 1, [2302].log_data[11].valid := 1,
        [2302].log_data[12].valid := 1, [2302].log_data[13].valid := 1, [2302].log_data[14].valid := 1, [2302].log_data[15].valid := 1, [2302].log_data[16].valid := 1, [2302].log_data[17].valid := 1, [2302].log_data[18].valid := 1, [2302].log_data[19].valid := 1, [2302].time.Year := 2023, [2302].time.Month := 1, [2302].time.Day := 17, [2302].time.Hour := 16, [2302].time.Minute := 14, [2302].time.Second := 59, [2303].log_data[0].min := 1.0, [2303].log_data[0].max := 1.0, [2303].log_data[0].total := 300.0, [2303].log_data[0].time := 300.0, [2303].log_data[0].minminute := 15, [2303].log_data[0].maxminute := 15, [2303].log_data[0].valid := 1, [2303].log_data[1].valid := 1, [2303].log_data[2].valid := 1, [2303].log_data[3].valid := 1, [2303].log_data[4].valid := 1, [2303].log_data[5].valid := 1, [2303].log_data[6].valid := 1, [2303].log_data[7].valid := 1, [2303].log_data[8].valid := 1, [2303].log_data[9].valid := 1, [2303].log_data[10].valid := 1, [2303].log_data[11].valid := 1, [2303].log_data[12].valid := 1, [2303].log_data[13].valid := 1, [2303].log_data[14].valid := 1, [2303].log_data[15].valid := 1, [2303].log_data[16].valid := 1, [2303].log_data[17].valid := 1, [2303].log_data[18].valid := 1, [2303].log_data[19].valid := 1, [2303].time.Year := 2023, [2303].time.Month := 1, [2303].time.Day := 17, [2303].time.Hour := 16, [2303].time.Minute := 19, [2303].time.Second := 59, [2304].log_data[0].min := 1.0, [2304].log_data[0].max := 1.0, [2304].log_data[0].total := 300.0, [2304].log_data[0].time := 300.0, [2304].log_data[0].minminute := 20, [2304].log_data[0].maxminute := 20, [2304].log_data[0].valid := 1, [2304].log_data[1].valid := 1, [2304].log_data[2].valid := 1, [2304].log_data[3].valid := 1, [2304].log_data[4].valid := 1, [2304].log_data[5].valid := 1, [2304].log_data[6].valid := 1, [2304].log_data[7].valid := 1,
        [2304].log_data[8].valid := 1, [2304].log_data[9].valid := 1, [2304].log_data[10].valid := 1, [2304].log_data[11].valid := 1, [2304].log_data[12].valid := 1, [2304].log_data[13].valid := 1, [2304].log_data[14].valid := 1, [2304].log_data[15].valid := 1, [2304].log_data[16].valid := 1, [2304].log_data[17].valid := 1, [2304].log_data[18].valid := 1, [2304].log_data[19].valid := 1, [2304].time.Year := 2023, [2304].time.Month := 1, [2304].time.Day := 17, [2304].time.Hour := 16, [2304].time.Minute := 24, [2304].time.Second := 59, [2305].log_data[0].min := 1.0, [2305].log_data[0].max := 1.0, [2305].log_data[0].total := 300.0, [2305].log_data[0].time := 300.0, [2305].log_data[0].minminute := 25, [2305].log_data[0].maxminute := 25, [2305].log_data[0].valid := 1, [2305].log_data[1].valid := 1, [2305].log_data[2].valid := 1, [2305].log_data[3].valid := 1, [2305].log_data[4].valid := 1, [2305].log_data[5].valid := 1, [2305].log_data[6].valid := 1, [2305].log_data[7].valid := 1, [2305].log_data[8].valid := 1, [2305].log_data[9].valid := 1, [2305].log_data[10].valid := 1, [2305].log_data[11].valid := 1, [2305].log_data[12].valid := 1, [2305].log_data[13].valid := 1, [2305].log_data[14].valid := 1, [2305].log_data[15].valid := 1, [2305].log_data[16].valid := 1, [2305].log_data[17].valid := 1, [2305].log_data[18].valid := 1, [2305].log_data[19].valid := 1, [2305].time.Year := 2023, [2305].time.Month := 1, [2305].time.Day := 17, [2305].time.Hour := 16, [2305].time.Minute := 29, [2305].time.Second := 59, [2306].log_data[0].min := 1.0, [2306].log_data[0].max := 1.0, [2306].log_data[0].total := 300.0, [2306].log_data[0].time := 300.0, [2306].log_data[0].minminute := 30, [2306].log_data[0].maxminute := 30, [2306].log_data[0].valid := 1, [2306].log_data[1].valid := 1, [2306].log_data[2].valid := 1, [2306].log_data[3].valid := 1,
        [2306].log_data[4].valid := 1, [2306].log_data[5].valid := 1, [2306].log_data[6].valid := 1, [2306].log_data[7].valid := 1, [2306].log_data[8].valid := 1, [2306].log_data[9].valid := 1, [2306].log_data[10].valid := 1, [2306].log_data[11].valid := 1, [2306].log_data[12].valid := 1, [2306].log_data[13].valid := 1, [2306].log_data[14].valid := 1, [2306].log_data[15].valid := 1, [2306].log_data[16].valid := 1, [2306].log_data[17].valid := 1, [2306].log_data[18].valid := 1, [2306].log_data[19].valid := 1, [2306].time.Year := 2023, [2306].time.Month := 1, [2306].time.Day := 17, [2306].time.Hour := 16, [2306].time.Minute := 34, [2306].time.Second := 59, [2307].log_data[0].min := 1.0, [2307].log_data[0].max := 1.0, [2307].log_data[0].total := 300.0, [2307].log_data[0].time := 300.0, [2307].log_data[0].minminute := 35, [2307].log_data[0].maxminute := 35, [2307].log_data[0].valid := 1, [2307].log_data[1].valid := 1, [2307].log_data[2].valid := 1, [2307].log_data[3].valid := 1, [2307].log_data[4].valid := 1, [2307].log_data[5].valid := 1, [2307].log_data[6].valid := 1, [2307].log_data[7].valid := 1, [2307].log_data[8].valid := 1, [2307].log_data[9].valid := 1, [2307].log_data[10].valid := 1, [2307].log_data[11].valid := 1, [2307].log_data[12].valid := 1, [2307].log_data[13].valid := 1, [2307].log_data[14].valid := 1, [2307].log_data[15].valid := 1, [2307].log_data[16].valid := 1, [2307].log_data[17].valid := 1, [2307].log_data[18].valid := 1, [2307].log_data[19].valid := 1, [2307].time.Year := 2023, [2307].time.Month := 1, [2307].time.Day := 17, [2307].time.Hour := 16, [2307].time.Minute := 39, [2307].time.Second := 59, [2308].log_data[0].min := 1.0, [2308].log_data[0].max := 1.0, [2308].log_data[0].total := 300.0, [2308].log_data[0].time := 300.0, [2308].log_data[0].minminute := 40, [2308].log_data[0].maxminute := 40,
        [2308].log_data[0].valid := 1, [2308].log_data[1].valid := 1, [2308].log_data[2].valid := 1, [2308].log_data[3].valid := 1, [2308].log_data[4].valid := 1, [2308].log_data[5].valid := 1, [2308].log_data[6].valid := 1, [2308].log_data[7].valid := 1, [2308].log_data[8].valid := 1, [2308].log_data[9].valid := 1, [2308].log_data[10].valid := 1, [2308].log_data[11].valid := 1, [2308].log_data[12].valid := 1, [2308].log_data[13].valid := 1, [2308].log_data[14].valid := 1, [2308].log_data[15].valid := 1, [2308].log_data[16].valid := 1, [2308].log_data[17].valid := 1, [2308].log_data[18].valid := 1, [2308].log_data[19].valid := 1, [2308].time.Year := 2023, [2308].time.Month := 1, [2308].time.Day := 17, [2308].time.Hour := 16, [2308].time.Minute := 44, [2308].time.Second := 59, [2309].log_data[0].min := 1.0, [2309].log_data[0].max := 1.0, [2309].log_data[0].total := 300.0, [2309].log_data[0].time := 300.0, [2309].log_data[0].minminute := 45, [2309].log_data[0].maxminute := 45, [2309].log_data[0].valid := 1, [2309].log_data[1].valid := 1, [2309].log_data[2].valid := 1, [2309].log_data[3].valid := 1, [2309].log_data[4].valid := 1, [2309].log_data[5].valid := 1, [2309].log_data[6].valid := 1, [2309].log_data[7].valid := 1, [2309].log_data[8].valid := 1, [2309].log_data[9].valid := 1, [2309].log_data[10].valid := 1, [2309].log_data[11].valid := 1, [2309].log_data[12].valid := 1, [2309].log_data[13].valid := 1, [2309].log_data[14].valid := 1, [2309].log_data[15].valid := 1, [2309].log_data[16].valid := 1, [2309].log_data[17].valid := 1, [2309].log_data[18].valid := 1, [2309].log_data[19].valid := 1, [2309].time.Year := 2023, [2309].time.Month := 1, [2309].time.Day := 17, [2309].time.Hour := 16, [2309].time.Minute := 49, [2309].time.Second := 59, [2310].log_data[0].min := 1.0, [2310].log_data[0].max := 1.0,
        [2310].log_data[0].total := 300.0, [2310].log_data[0].time := 300.0, [2310].log_data[0].minminute := 50, [2310].log_data[0].maxminute := 50, [2310].log_data[0].valid := 1, [2310].log_data[1].valid := 1, [2310].log_data[2].valid := 1, [2310].log_data[3].valid := 1, [2310].log_data[4].valid := 1, [2310].log_data[5].valid := 1, [2310].log_data[6].valid := 1, [2310].log_data[7].valid := 1, [2310].log_data[8].valid := 1, [2310].log_data[9].valid := 1, [2310].log_data[10].valid := 1, [2310].log_data[11].valid := 1, [2310].log_data[12].valid := 1, [2310].log_data[13].valid := 1, [2310].log_data[14].valid := 1, [2310].log_data[15].valid := 1, [2310].log_data[16].valid := 1, [2310].log_data[17].valid := 1, [2310].log_data[18].valid := 1, [2310].log_data[19].valid := 1, [2310].time.Year := 2023, [2310].time.Month := 1, [2310].time.Day := 17, [2310].time.Hour := 16, [2310].time.Minute := 54, [2310].time.Second := 59, [2311].log_data[0].min := 1.0, [2311].log_data[0].max := 1.0, [2311].log_data[0].total := 300.0, [2311].log_data[0].time := 300.0, [2311].log_data[0].minminute := 55, [2311].log_data[0].maxminute := 55, [2311].log_data[0].valid := 1, [2311].log_data[1].valid := 1, [2311].log_data[2].valid := 1, [2311].log_data[3].valid := 1, [2311].log_data[4].valid := 1, [2311].log_data[5].valid := 1, [2311].log_data[6].valid := 1, [2311].log_data[7].valid := 1, [2311].log_data[8].valid := 1, [2311].log_data[9].valid := 1, [2311].log_data[10].valid := 1, [2311].log_data[11].valid := 1, [2311].log_data[12].valid := 1, [2311].log_data[13].valid := 1, [2311].log_data[14].valid := 1, [2311].log_data[15].valid := 1, [2311].log_data[16].valid := 1, [2311].log_data[17].valid := 1, [2311].log_data[18].valid := 1, [2311].log_data[19].valid := 1, [2311].time.Year := 2023, [2311].time.Month := 1, [2311].time.Day := 17, [2311].time.Hour := 16,
        [2311].time.Minute := 59, [2311].time.Second := 59, [2312].log_data[0].min := 1.0, [2312].log_data[0].max := 1.0, [2312].log_data[0].total := 300.0, [2312].log_data[0].time := 300.0, [2312].log_data[0].valid := 1, [2312].log_data[1].valid := 1, [2312].log_data[2].valid := 1, [2312].log_data[3].valid := 1, [2312].log_data[4].valid := 1, [2312].log_data[5].valid := 1, [2312].log_data[6].valid := 1, [2312].log_data[7].valid := 1, [2312].log_data[8].valid := 1, [2312].log_data[9].valid := 1, [2312].log_data[10].valid := 1, [2312].log_data[11].valid := 1, [2312].log_data[12].valid := 1, [2312].log_data[13].valid := 1, [2312].log_data[14].valid := 1, [2312].log_data[15].valid := 1, [2312].log_data[16].valid := 1, [2312].log_data[17].valid := 1, [2312].log_data[18].valid := 1, [2312].log_data[19].valid := 1, [2312].time.Year := 2023, [2312].time.Month := 1, [2312].time.Day := 17, [2312].time.Hour := 17, [2312].time.Minute := 4, [2312].time.Second := 59, [2313].log_data[0].min := 1.0, [2313].log_data[0].max := 1.0, [2313].log_data[0].total := 300.0, [2313].log_data[0].time := 300.0, [2313].log_data[0].minminute := 5, [2313].log_data[0].maxminute := 5, [2313].log_data[0].valid := 1, [2313].log_data[1].valid := 1, [2313].log_data[2].valid := 1, [2313].log_data[3].valid := 1, [2313].log_data[4].valid := 1, [2313].log_data[5].valid := 1, [2313].log_data[6].valid := 1, [2313].log_data[7].valid := 1, [2313].log_data[8].valid := 1, [2313].log_data[9].valid := 1, [2313].log_data[10].valid := 1, [2313].log_data[11].valid := 1, [2313].log_data[12].valid := 1, [2313].log_data[13].valid := 1, [2313].log_data[14].valid := 1, [2313].log_data[15].valid := 1, [2313].log_data[16].valid := 1, [2313].log_data[17].valid := 1, [2313].log_data[18].valid := 1, [2313].log_data[19].valid := 1, [2313].time.Year := 2023, [2313].time.Month := 1,
        [2313].time.Day := 17, [2313].time.Hour := 17, [2313].time.Minute := 9, [2313].time.Second := 59, [2314].log_data[0].min := 1.0, [2314].log_data[0].max := 1.0, [2314].log_data[0].total := 300.0, [2314].log_data[0].time := 300.0, [2314].log_data[0].minminute := 10, [2314].log_data[0].maxminute := 10, [2314].log_data[0].valid := 1, [2314].log_data[1].valid := 1, [2314].log_data[2].valid := 1, [2314].log_data[3].valid := 1, [2314].log_data[4].valid := 1, [2314].log_data[5].valid := 1, [2314].log_data[6].valid := 1, [2314].log_data[7].valid := 1, [2314].log_data[8].valid := 1, [2314].log_data[9].valid := 1, [2314].log_data[10].valid := 1, [2314].log_data[11].valid := 1, [2314].log_data[12].valid := 1, [2314].log_data[13].valid := 1, [2314].log_data[14].valid := 1, [2314].log_data[15].valid := 1, [2314].log_data[16].valid := 1, [2314].log_data[17].valid := 1, [2314].log_data[18].valid := 1, [2314].log_data[19].valid := 1, [2314].time.Year := 2023, [2314].time.Month := 1, [2314].time.Day := 17, [2314].time.Hour := 17, [2314].time.Minute := 14, [2314].time.Second := 59, [2315].log_data[0].min := 1.0, [2315].log_data[0].max := 1.0, [2315].log_data[0].total := 300.0, [2315].log_data[0].time := 300.0, [2315].log_data[0].minminute := 15, [2315].log_data[0].maxminute := 15, [2315].log_data[0].valid := 1, [2315].log_data[1].valid := 1, [2315].log_data[2].valid := 1, [2315].log_data[3].valid := 1, [2315].log_data[4].valid := 1, [2315].log_data[5].valid := 1, [2315].log_data[6].valid := 1, [2315].log_data[7].valid := 1, [2315].log_data[8].valid := 1, [2315].log_data[9].valid := 1, [2315].log_data[10].valid := 1, [2315].log_data[11].valid := 1, [2315].log_data[12].valid := 1, [2315].log_data[13].valid := 1, [2315].log_data[14].valid := 1, [2315].log_data[15].valid := 1, [2315].log_data[16].valid := 1, [2315].log_data[17].valid := 1,
        [2315].log_data[18].valid := 1, [2315].log_data[19].valid := 1, [2315].time.Year := 2023, [2315].time.Month := 1, [2315].time.Day := 17, [2315].time.Hour := 17, [2315].time.Minute := 19, [2315].time.Second := 59, [2316].log_data[0].min := 1.0, [2316].log_data[0].max := 1.0, [2316].log_data[0].total := 300.0, [2316].log_data[0].time := 300.0, [2316].log_data[0].minminute := 20, [2316].log_data[0].maxminute := 20, [2316].log_data[0].valid := 1, [2316].log_data[1].valid := 1, [2316].log_data[2].valid := 1, [2316].log_data[3].valid := 1, [2316].log_data[4].valid := 1, [2316].log_data[5].valid := 1, [2316].log_data[6].valid := 1, [2316].log_data[7].valid := 1, [2316].log_data[8].valid := 1, [2316].log_data[9].valid := 1, [2316].log_data[10].valid := 1, [2316].log_data[11].valid := 1, [2316].log_data[12].valid := 1, [2316].log_data[13].valid := 1, [2316].log_data[14].valid := 1, [2316].log_data[15].valid := 1, [2316].log_data[16].valid := 1, [2316].log_data[17].valid := 1, [2316].log_data[18].valid := 1, [2316].log_data[19].valid := 1, [2316].time.Year := 2023, [2316].time.Month := 1, [2316].time.Day := 17, [2316].time.Hour := 17, [2316].time.Minute := 24, [2316].time.Second := 59, [2317].log_data[0].min := 1.0, [2317].log_data[0].max := 1.0, [2317].log_data[0].total := 300.0, [2317].log_data[0].time := 300.0, [2317].log_data[0].minminute := 25, [2317].log_data[0].maxminute := 25, [2317].log_data[0].valid := 1, [2317].log_data[1].valid := 1, [2317].log_data[2].valid := 1, [2317].log_data[3].valid := 1, [2317].log_data[4].valid := 1, [2317].log_data[5].valid := 1, [2317].log_data[6].valid := 1, [2317].log_data[7].valid := 1, [2317].log_data[8].valid := 1, [2317].log_data[9].valid := 1, [2317].log_data[10].valid := 1, [2317].log_data[11].valid := 1, [2317].log_data[12].valid := 1, [2317].log_data[13].valid := 1,
        [2317].log_data[14].valid := 1, [2317].log_data[15].valid := 1, [2317].log_data[16].valid := 1, [2317].log_data[17].valid := 1, [2317].log_data[18].valid := 1, [2317].log_data[19].valid := 1, [2317].time.Year := 2023, [2317].time.Month := 1, [2317].time.Day := 17, [2317].time.Hour := 17, [2317].time.Minute := 29, [2317].time.Second := 59, [2318].log_data[0].min := 1.0, [2318].log_data[0].max := 1.0, [2318].log_data[0].total := 300.0, [2318].log_data[0].time := 300.0, [2318].log_data[0].minminute := 30, [2318].log_data[0].maxminute := 30, [2318].log_data[0].valid := 1, [2318].log_data[1].valid := 1, [2318].log_data[2].valid := 1, [2318].log_data[3].valid := 1, [2318].log_data[4].valid := 1, [2318].log_data[5].valid := 1, [2318].log_data[6].valid := 1, [2318].log_data[7].valid := 1, [2318].log_data[8].valid := 1, [2318].log_data[9].valid := 1, [2318].log_data[10].valid := 1, [2318].log_data[11].valid := 1, [2318].log_data[12].valid := 1, [2318].log_data[13].valid := 1, [2318].log_data[14].valid := 1, [2318].log_data[15].valid := 1, [2318].log_data[16].valid := 1, [2318].log_data[17].valid := 1, [2318].log_data[18].valid := 1, [2318].log_data[19].valid := 1, [2318].time.Year := 2023, [2318].time.Month := 1, [2318].time.Day := 17, [2318].time.Hour := 17, [2318].time.Minute := 34, [2318].time.Second := 59, [2319].log_data[0].min := 1.0, [2319].log_data[0].max := 1.0, [2319].log_data[0].total := 300.0, [2319].log_data[0].time := 300.0, [2319].log_data[0].minminute := 35, [2319].log_data[0].maxminute := 35, [2319].log_data[0].valid := 1, [2319].log_data[1].valid := 1, [2319].log_data[2].valid := 1, [2319].log_data[3].valid := 1, [2319].log_data[4].valid := 1, [2319].log_data[5].valid := 1, [2319].log_data[6].valid := 1, [2319].log_data[7].valid := 1, [2319].log_data[8].valid := 1, [2319].log_data[9].valid := 1,
